  MoveL 1319 to (26.76, 68.08, -94.98) mm, rotated rx -9.61 ry -16.54 rz 125.97 deg; joints [-8.897, -67.323, 117.954, 201.647, 36.046, -119.29, -235]
  MoveL 1320 to (26.41, 68.69, -94.98) mm, rotated rx -9.61 ry -16.54 rz 125.97 deg; joints [-8.899, -67.37, 118.001, 201.644, 36.045, -119.288, -235]
  MoveL 1321 to (26.18, 69.29, -94.97) mm, rotated rx -9.61 ry -16.54 rz 125.97 deg; joints [-8.9, -67.415, 118.038, 201.646, 36.038, -119.292, -235]
  MoveL 1322 to (25.98, 69.92, -94.95) mm, rotated rx -9.61 ry -16.54 rz 125.97 deg; joints [-8.901, -67.462, 118.074, 201.65, 36.028, -119.298, -235]
  MoveL 1323 to (25.77, 70.66, -94.92) mm, rotated rx -9.61 ry -16.54 rz 125.97 deg; joints [-8.902, -67.516, 118.114, 201.657, 36.015, -119.306, -235]
  MoveL 1324 to (25.28, 72.7, -94.92) mm, rotated rx -9.61 ry -16.54 rz 125.97 deg; joints [-8.906, -67.664, 118.218, 201.672, 35.972, -119.329, -235]
  MoveL 1325 to (25.17, 73.13, -94.9) mm, rotated rx -9.61 ry -16.54 rz 125.97 deg; joints [-8.907, -67.696, 118.241, 201.676, 35.964, -119.335, -235]
  MoveL 1326 to (24.92, 74.15, -94.9) mm, rotated rx -9.61 ry -16.54 rz 125.97 deg; joints [-8.909, -67.77, 118.292, 201.684, 35.942, -119.347, -235]
  MoveL 1327 to (24.8, 74.64, -94.89) mm, rotated rx -9.61 ry -16.54 rz 125.97 deg; joints [-8.91, -67.806, 118.318, 201.688, 35.932, -119.352, -235]
  MoveL 1328 to (24.68, 75.11, -94.87) mm, rotated rx -9.61 ry -16.54 rz 125.97 deg; joints [-8.91, -67.841, 118.343, 201.692, 35.923, -119.358, -235]
  MoveL 1329 to (24.54, 75.57, -94.84) mm, rotated rx -9.61 ry -16.54 rz 125.97 deg; joints [-8.91, -67.875, 118.368, 201.697, 35.915, -119.364, -235]
  MoveL 1330 to (24.4, 75.98, -94.78) mm, rotated rx -9.61 ry -16.54 rz 125.97 deg; joints [-8.909, -67.906, 118.392, 201.703, 35.909, -119.37, -235]
  MoveL 1331 to (24.27, 76.44, -94.75) mm, rotated rx -9.61 ry -16.54 rz 125.97 deg; joints [-8.908, -67.939, 118.417, 201.708, 35.901, -119.376, -235]
  MoveL 1332 to (24.14, 76.91, -94.73) mm, rotated rx -9.61 ry -16.54 rz 125.97 deg; joints [-8.908, -67.974, 118.442, 201.712, 35.892, -119.381, -235]
  MoveL 1333 to (24.02, 77.41, -94.72) mm, rotated rx -9.61 ry -16.54 rz 125.97 deg; joints [-8.909, -68.01, 118.468, 201.717, 35.882, -119.387, -235]
  MoveL 1334 to (23.89, 77.88, -94.7) mm, rotated rx -9.61 ry -16.54 rz 125.97 deg; joints [-8.91, -68.045, 118.493, 201.721, 35.873, -119.393, -235]
  MoveL 1335 to (23.75, 78.34, -94.67) mm, rotated rx -9.61 ry -16.54 rz 125.97 deg; joints [-8.909, -68.079, 118.518, 201.726, 35.865, -119.399, -235]
  MoveL 1336 to (23.61, 78.75, -94.61) mm, rotated rx -9.61 ry -16.54 rz 125.97 deg; joints [-8.908, -68.11, 118.543, 201.731, 35.859, -119.404, -235]
  MoveL 1337 to (23.46, 79.18, -94.55) mm, rotated rx -9.61 ry -16.54 rz 125.97 deg; joints [-8.907, -68.143, 118.568, 201.737, 35.853, -119.41, -235]
  MoveL 1338 to (23.06, 80.57, -94.47) mm, rotated rx -9.61 ry -16.54 rz 125.97 deg; joints [-8.906, -68.245, 118.644, 201.751, 35.828, -119.427, -235]
  MoveL 1339 to (22.88, 81.73, -94.6) mm, rotated rx -9.61 ry -16.54 rz 125.97 deg; joints [-8.914, -68.328, 118.694, 201.755, 35.796, -119.44, -235]
  MoveL 1340 to (22.91, 82.67, -94.94) mm, rotated rx -9.61 ry -16.54 rz 125.97 deg; joints [-8.931, -68.392, 118.719, 201.749, 35.756, -119.448, -235]
  MoveL 1341 to (23.01, 83.06, -95.18) mm, rotated rx -9.61 ry -16.54 rz 125.97 deg; joints [-8.942, -68.416, 118.722, 201.742, 35.733, -119.45, -235]
  MoveL 1342 to (23.16, 83.39, -95.48) mm, rotated rx -9.61 ry -16.54 rz 125.97 deg; joints [-8.955, -68.436, 118.719, 201.733, 35.709, -119.451, -235]
  MoveL 1343 to (23.62, 83.9, -96.24) mm, rotated rx -9.61 ry -16.54 rz 125.97 deg; joints [-8.988, -68.461, 118.694, 201.706, 35.655, -119.449, -235]
  MoveL 1344 to (24.31, 84.18, -97.21) mm, rotated rx -9.61 ry -16.54 rz 125.97 deg; joints [-9.029, -68.466, 118.644, 201.669, 35.593, -119.443, -235]
  MoveL 1345 to (26.32, 84.09, -99.77) mm, rotated rx -9.61 ry -16.54 rz 125.97 deg; joints [-9.136, -68.419, 118.468, 201.565, 35.449, -119.415, -235]
  MoveL 1346 to (28.5, 83.24, -102.39) mm, rotated rx -9.61 ry -16.54 rz 125.97 deg; joints [-9.242, -68.314, 118.254, 201.451, 35.322, -119.375, -235]
  MoveL 1347 to (29.39, 82.56, -103.41) mm, rotated rx -9.61 ry -16.54 rz 125.97 deg; joints [-9.283, -68.249, 118.156, 201.402, 35.281, -119.353, -235]
  MoveL 1348 to (30.16, 81.72, -104.25) mm, rotated rx -9.61 ry -16.54 rz 125.97 deg; joints [-9.315, -68.176, 118.064, 201.358, 35.257, -119.33, -235]
  MoveL 1349 to (30.79, 80.72, -104.9) mm, rotated rx -9.61 ry -16.54 rz 125.97 deg; joints [-9.34, -68.094, 117.979, 201.32, 35.248, -119.307, -235]
  MoveL 1350 to (31.3, 79.55, -105.37) mm, rotated rx -9.61 ry -16.54 rz 125.97 deg; joints [-9.357, -68.004, 117.899, 201.288, 35.254, -119.283, -235]
  MoveL 1351 to (31.67, 78.22, -105.65) mm, rotated rx -9.61 ry -16.54 rz 125.97 deg; joints [-9.365, -67.905, 117.826, 201.261, 35.276, -119.258, -235]
  MoveL 1352 to (31.92, 76.73, -105.74) mm, rotated rx -9.61 ry -16.54 rz 125.97 deg; joints [-9.366, -67.798, 117.759, 201.239, 35.313, -119.232, -235]
  MoveL 1353 to (32.27, 73.59, -105.75) mm, rotated rx -9.61 ry -16.54 rz 125.97 deg; joints [-9.359, -67.576, 117.631, 201.203, 35.402, -119.181, -235]
  MoveL 1354 to (32.34, 73.04, -105.76) mm, rotated rx -9.61 ry -16.54 rz 125.97 deg; joints [-9.358, -67.537, 117.608, 201.196, 35.417, -119.172, -235]
  MoveL 1355 to (32.44, 72.42, -105.8) mm, rotated rx -9.61 ry -16.54 rz 125.97 deg; joints [-9.358, -67.493, 117.58, 201.187, 35.432, -119.161, -235]
  MoveL 1356 to (32.58, 71.68, -105.89) mm, rotated rx -9.61 ry -16.54 rz 125.97 deg; joints [-9.361, -67.439, 117.544, 201.174, 35.449, -119.148, -235]
  MoveL 1357 to (32.68, 71.07, -105.93) mm, rotated rx -9.61 ry -16.54 rz 125.97 deg; joints [-9.361, -67.395, 117.517, 201.166, 35.464, -119.137, -235]
  MoveL 1358 to (32.75, 70.53, -105.94) mm, rotated rx -9.61 ry -16.54 rz 125.97 deg; joints [-9.36, -67.357, 117.494, 201.159, 35.478, -119.128, -235]
  MoveL 1359 to (32.81, 70.02, -105.95) mm, rotated rx -9.61 ry -16.54 rz 125.97 deg; joints [-9.36, -67.321, 117.473, 201.153, 35.492, -119.12, -235]
  MoveL 1360 to (32.88, 69.57, -105.97) mm, rotated rx -9.61 ry -16.54 rz 125.97 deg; joints [-9.359, -67.289, 117.453, 201.147, 35.504, -119.113, -235]
  MoveL 1361 to (33.12, 67.53, -105.97) mm, rotated rx -9.61 ry -16.54 rz 125.97 deg; joints [-9.355, -67.145, 117.368, 201.124, 35.56, -119.08, -235]
  MoveL 1362 to (33.2, 67.02, -106.01) mm, rotated rx -9.61 ry -16.54 rz 125.97 deg; joints [-9.355, -67.109, 117.345, 201.117, 35.572, -119.072, -235]
  MoveL 1363 to (33.29, 66.56, -106.06) mm, rotated rx -9.61 ry -16.54 rz 125.97 deg; joints [-9.356, -67.075, 117.323, 201.109, 35.582, -119.064, -235]
  MoveL 1364 to (33.39, 66.11, -106.13) mm, rotated rx -9.61 ry -16.54 rz 125.97 deg; joints [-9.358, -67.042, 117.299, 201.101, 35.591, -119.056, -235]
  MoveL 1365 to (33.53, 65.64, -106.19) mm, rotated rx -9.61 ry -16.54 rz 125.97 deg; joints [-9.36, -67.008, 117.273, 201.095, 35.598, -119.049, -235]
  MoveL 1366 to (33.69, 65.11, -106.23) mm, rotated rx -9.61 ry -16.54 rz 125.97 deg; joints [-9.36, -66.969, 117.243, 201.091, 35.606, -119.044, -235]
  MoveL 1367 to (33.98, 64.51, -106.24) mm, rotated rx -9.61 ry -16.54 rz 125.97 deg; joints [-9.358, -66.923, 117.2, 201.092, 35.61, -119.043, -235]
  MoveL 1368 to (34.38, 63.84, -106.24) mm, rotated rx -9.61 ry -16.54 rz 125.97 deg; joints [-9.356, -66.871, 117.148, 201.096, 35.61, -119.046, -235]
  MoveL 1369 to (34.29, 65.78, -107.79) mm, rotated rx -9.61 ry -16.54 rz 125.97 deg; joints [-9.427, -66.999, 117.207, 201.017, 35.529, -119.016, -235]
  MoveL 1370 to (35.84, 64, -107.92) mm, rotated rx -9.61 ry -16.54 rz 125.97 deg; joints [-9.424, -66.852, 117.027, 201.037, 35.499, -119.039, -235]
  MoveL 1371 to (37.3, 62.31, -108.03) mm, rotated rx -9.61 ry -16.54 rz 125.97 deg; joints [-9.421, -66.713, 116.857, 201.058, 35.471, -119.061, -235]
  MoveL 1372 to (38.73, 60.68, -108.19) mm, rotated rx -9.61 ry -16.54 rz 125.97 deg; joints [-9.42, -66.579, 116.692, 201.075, 35.442, -119.082, -235]
  MoveL 1373 to (40.12, 59.07, -108.3) mm, rotated rx -9.61 ry -16.54 rz 125.97 deg; joints [-9.418, -66.446, 116.529, 201.095, 35.414, -119.103, -235]
  MoveL 1374 to (41.52, 57.45, -108.41) mm, rotated rx -9.61 ry -16.54 rz 125.97 deg; joints [-9.415, -66.313, 116.365, 201.114, 35.386, -119.125, -235]
  MoveL 1375 to (42.92, 55.84, -108.63) mm, rotated rx -9.61 ry -16.54 rz 125.97 deg; joints [-9.417, -66.181, 116.201, 201.127, 35.356, -119.143, -235]
  MoveL 1376 to (44.32, 54.23, -108.86) mm, rotated rx -9.61 ry -16.54 rz 125.97 deg; joints [-9.419, -66.048, 116.036, 201.14, 35.326, -119.16, -235]
  MoveL 1377 to (45.71, 52.61, -108.97) mm, rotated rx -9.61 ry -16.54 rz 125.97 deg; joints [-9.416, -65.915, 115.872, 201.16, 35.298, -119.182, -235]
  MoveL 1378 to (47.09, 50.98, -108.97) mm, rotated rx -9.61 ry -16.54 rz 125.97 deg; joints [-9.409, -65.782, 115.71, 201.187, 35.272, -119.209, -235]
  MoveL 1379 to (48.48, 49.36, -109.08) mm, rotated rx -9.61 ry -16.54 rz 125.97 deg; joints [-9.406, -65.65, 115.546, 201.207, 35.243, -119.231, -235]
  MoveL 1380 to (49.88, 47.71, -109.29) mm, rotated rx -9.61 ry -16.54 rz 125.97 deg; joints [-9.408, -65.515, 115.379, 201.222, 35.213, -119.25, -235]
  MoveL 1381 to (51.19, 46.18, -109.47) mm, rotated rx -9.61 ry -16.54 rz 125.97 deg; joints [-9.408, -65.389, 115.223, 201.236, 35.185, -119.268, -235]
  MoveL 1382 to (52.39, 44.76, -109.68) mm, rotated rx -9.61 ry -16.54 rz 125.97 deg; joints [-9.411, -65.273, 115.079, 201.246, 35.158, -119.282, -235]
  MoveL 1383 to (53.66, 43.26, -109.77) mm, rotated rx -9.61 ry -16.54 rz 125.97 deg; joints [-9.408, -65.151, 114.928, 201.266, 35.131, -119.304, -235]
  MoveL 1384 to (55.01, 41.67, -109.79) mm, rotated rx -9.61 ry -16.54 rz 125.97 deg; joints [-9.402, -65.021, 114.767, 201.292, 35.104, -119.331, -235]
  MoveL 1385 to (56.75, 39.59, -109.88) mm, rotated rx -9.61 ry -16.54 rz 125.97 deg; joints [-9.397, -64.853, 114.558, 201.322, 35.067, -119.361, -235]
  MoveL 1386 to (58.05, 38.03, -110.1) mm, rotated rx -9.61 ry -16.54 rz 125.97 deg; joints [-9.399, -64.725, 114.4, 201.334, 35.039, -119.378, -235]
  MoveL 1387 to (59.45, 36.33, -110.3) mm, rotated rx -9.61 ry -16.54 rz 125.97 deg; joints [-9.4, -64.587, 114.23, 201.349, 35.008, -119.398, -235]
  MoveL 1388 to (60.73, 34.76, -110.58) mm, rotated rx -9.61 ry -16.54 rz 125.97 deg; joints [-9.405, -64.46, 114.073, 201.356, 34.979, -119.411, -235]
  MoveL 1389 to (62, 33.24, -110.71) mm, rotated rx -9.61 ry -16.54 rz 125.97 deg; joints [-9.404, -64.336, 113.919, 201.374, 34.951, -119.432, -235]
  MoveL 1390 to (63.36, 31.64, -110.73) mm, rotated rx -9.61 ry -16.54 rz 125.97 deg; joints [-9.397, -64.207, 113.756, 201.402, 34.922, -119.46, -235]
  MoveL 1391 to (64.46, 30.25, -110.96) mm, rotated rx -9.61 ry -16.54 rz 125.97 deg; joints [-9.401, -64.095, 113.619, 201.409, 34.897, -119.472, -235]
  Set speed (1000.0 mm/s)
  MoveL 1392 to (88.08, 19.24, -110.96) mm, rotated rx -9.61 ry -16.54 rz 125.97 deg; joints [-9.309, -62.966, 111.351, 202.177, 33.862, -120.32, -235]
  Set speed (1000.0 mm/s)
  MoveL 1393 to (85.31, 13.32, -122.15) mm, rotated rx -9.61 ry -16.54 rz 125.97 deg; joints [-9.767, -62.572, 111.273, 201.243, 34.045, -119.606, -235]
  Set speed (100.0 mm/s)
  MoveL 1394 to (67.03, 21.84, -122.15) mm, rotated rx -9.61 ry -16.54 rz 125.97 deg; joints [-9.843, -63.44, 113.032, 200.653, 34.858, -118.961, -235]
  MoveL 1395 to (65.87, 23.63, -122.15) mm, rotated rx -9.61 ry -16.54 rz 125.97 deg; joints [-9.851, -63.579, 113.188, 200.632, 34.872, -118.942, -235]
  MoveL 1396 to (64.67, 25.51, -122.05) mm, rotated rx -9.61 ry -16.54 rz 125.97 deg; joints [-9.855, -63.725, 113.35, 200.618, 34.886, -118.929, -235]
  MoveL 1397 to (63.44, 27.51, -121.75) mm, rotated rx -9.61 ry -16.54 rz 125.97 deg; joints [-9.85, -63.88, 113.52, 200.617, 34.901, -118.924, -235]
  MoveL 1398 to (62.26, 29.43, -121.41) mm, rotated rx -9.61 ry -16.54 rz 125.97 deg; joints [-9.844, -64.03, 113.683, 200.621, 34.915, -118.923, -235]
  MoveL 1399 to (61.15, 31.18, -121.22) mm, rotated rx -9.61 ry -16.54 rz 125.97 deg; joints [-9.843, -64.166, 113.833, 200.616, 34.928, -118.915, -235]
  MoveL 1400 to (60.1, 32.82, -121.08) mm, rotated rx -9.61 ry -16.54 rz 125.97 deg; joints [-9.844, -64.294, 113.974, 200.607, 34.941, -118.906, -235]
  MoveL 1401 to (58.98, 34.54, -121.03) mm, rotated rx -9.61 ry -16.54 rz 125.97 deg; joints [-9.849, -64.428, 114.123, 200.592, 34.953, -118.892, -235]
  MoveL 1402 to (57.82, 36.33, -121.01) mm, rotated rx -9.61 ry -16.54 rz 125.97 deg; joints [-9.856, -64.567, 114.277, 200.573, 34.965, -118.876, -235]
  MoveL 1403 to (56.66, 38.11, -120.89) mm, rotated rx -9.61 ry -16.54 rz 125.97 deg; joints [-9.858, -64.706, 114.43, 200.562, 34.978, -118.864, -235]
  MoveL 1404 to (55.42, 40.03, -120.63) mm, rotated rx -9.61 ry -16.54 rz 125.97 deg; joints [-9.856, -64.857, 114.596, 200.559, 34.992, -118.858, -235]
  MoveL 1405 to (54.1, 42.04, -120.45) mm, rotated rx -9.61 ry -16.54 rz 125.97 deg; joints [-9.856, -65.015, 114.769, 200.55, 35.007, -118.847, -235]
  MoveL 1406 to (52.82, 43.99, -120.25) mm, rotated rx -9.61 ry -16.54 rz 125.97 deg; joints [-9.856, -65.168, 114.938, 200.543, 35.022, -118.838, -235]
  MoveL 1407 to (51.65, 45.77, -120.13) mm, rotated rx -9.61 ry -16.54 rz 125.97 deg; joints [-9.859, -65.308, 115.092, 200.531, 35.034, -118.827, -235]
  MoveL 1408 to (49.32, 49.29, -119.86) mm, rotated rx -9.61 ry -16.54 rz 125.97 deg; joints [-9.862, -65.585, 115.396, 200.512, 35.058, -118.807, -235]
  MoveL 1409 to (48.13, 51.11, -119.79) mm, rotated rx -9.61 ry -16.54 rz 125.97 deg; joints [-9.867, -65.728, 115.551, 200.498, 35.068, -118.794, -235]
  MoveL 1410 to (46.94, 52.88, -119.57) mm, rotated rx -9.61 ry -16.54 rz 125.97 deg; joints [-9.866, -65.868, 115.705, 200.494, 35.082, -118.787, -235]
  MoveL 1411 to (45.76, 54.63, -119.41) mm, rotated rx -9.61 ry -16.54 rz 125.97 deg; joints [-9.866, -66.007, 115.857, 200.486, 35.094, -118.778, -235]
  MoveL 1412 to (44.58, 56.38, -119.23) mm, rotated rx -9.61 ry -16.54 rz 125.97 deg; joints [-9.866, -66.146, 116.009, 200.479, 35.107, -118.77, -235]
  MoveL 1413 to (43.37, 58.2, -119.14) mm, rotated rx -9.61 ry -16.54 rz 125.97 deg; joints [-9.87, -66.289, 116.164, 200.467, 35.117, -118.759, -235]
  MoveL 1414 to (42.1, 60.08, -119.01) mm, rotated rx -9.61 ry -16.54 rz 125.97 deg; joints [-9.873, -66.438, 116.327, 200.456, 35.13, -118.748, -235]
  MoveL 1415 to (41.06, 61.67, -118.95) mm, rotated rx -9.61 ry -16.54 rz 125.97 deg; joints [-9.877, -66.564, 116.461, 200.445, 35.136, -118.738, -235]
  MoveL 1416 to (40.5, 61.31, -118.06) mm, rotated rx -9.61 ry -16.54 rz 125.97 deg; joints [-9.84, -66.551, 116.499, 200.479, 35.192, -118.746, -235]
  MoveL 1417 to (40.48, 60.95, -117.65) mm, rotated rx -9.61 ry -16.54 rz 125.97 deg; joints [-9.822, -66.529, 116.492, 200.502, 35.21, -118.756, -235]
  MoveL 1418 to (40.44, 60.9, -117.37) mm, rotated rx -9.61 ry -16.54 rz 125.97 deg; joints [-9.81, -66.527, 116.496, 200.518, 35.218, -118.765, -235]
  MoveL 1419 to (40.39, 61.22, -117.26) mm, rotated rx -9.61 ry -16.54 rz 125.97 deg; joints [-9.806, -66.551, 116.511, 200.529, 35.212, -118.774, -235]
  MoveL 1420 to (40.36, 61.67, -117.19) mm, rotated rx -9.61 ry -16.54 rz 125.97 deg; joints [-9.804, -66.582, 116.529, 200.538, 35.199, -118.785, -235]
  MoveL 1421 to (40.34, 62.23, -117.16) mm, rotated rx -9.61 ry -16.54 rz 125.97 deg; joints [-9.804, -66.621, 116.549, 200.548, 35.182, -118.796, -235]
  MoveL 1422 to (40.33, 62.93, -117.12) mm, rotated rx -9.61 ry -16.54 rz 125.97 deg; joints [-9.804, -66.669, 116.574, 200.56, 35.16, -118.811, -235]
  MoveL 1423 to (40.32, 63.56, -117.1) mm, rotated rx -9.61 ry -16.54 rz 125.97 deg; joints [-9.804, -66.712, 116.595, 200.571, 35.139, -118.824, -235]
  MoveL 1424 to (40.33, 64.08, -117.1) mm, rotated rx -9.61 ry -16.54 rz 125.97 deg; joints [-9.805, -66.748, 116.612, 200.579, 35.121, -118.835, -235]
  MoveL 1425 to (40.32, 64.57, -117.08) mm, rotated rx -9.61 ry -16.54 rz 125.97 deg; joints [-9.805, -66.782, 116.628, 200.587, 35.105, -118.845, -235]
  MoveL 1426 to (40.28, 65.61, -117) mm, rotated rx -9.61 ry -16.54 rz 125.97 deg; joints [-9.804, -66.854, 116.666, 200.606, 35.073, -118.867, -235]
  MoveL 1427 to (40.25, 66.17, -116.95) mm, rotated rx -9.61 ry -16.54 rz 125.97 deg; joints [-9.803, -66.893, 116.687, 200.616, 35.056, -118.879, -235]
  MoveL 1428 to (40.21, 66.68, -116.89) mm, rotated rx -9.61 ry -16.54 rz 125.97 deg; joints [-9.802, -66.928, 116.707, 200.627, 35.042, -118.89, -235]
  MoveL 1429 to (40.17, 67.14, -116.81) mm, rotated rx -9.61 ry -16.54 rz 125.97 deg; joints [-9.8, -66.961, 116.726, 200.637, 35.03, -118.901, -235]
  MoveL 1430 to (40.14, 67.6, -116.75) mm, rotated rx -9.61 ry -16.54 rz 125.97 deg; joints [-9.798, -66.994, 116.744, 200.647, 35.016, -118.911, -235]
  MoveL 1431 to (40.12, 68.09, -116.72) mm, rotated rx -9.61 ry -16.54 rz 125.97 deg; joints [-9.798, -67.027, 116.761, 200.655, 35.001, -118.922, -235]
  MoveL 1432 to (40.11, 68.61, -116.7) mm, rotated rx -9.61 ry -16.54 rz 125.97 deg; joints [-9.798, -67.063, 116.779, 200.664, 34.984, -118.933, -235]
  MoveL 1433 to (40.15, 72.28, -116.7) mm, rotated rx -9.61 ry -16.54 rz 125.97 deg; joints [-9.805, -67.313, 116.893, 200.721, 34.856, -119.009, -235]
  MoveL 1434 to (40.28, 73.9, -116.72) mm, rotated rx -9.61 ry -16.54 rz 125.97 deg; joints [-9.809, -67.422, 116.935, 200.749, 34.792, -119.046, -235]
  MoveL 1435 to (40.42, 74.46, -116.75) mm, rotated rx -9.61 ry -16.54 rz 125.97 deg; joints [-9.811, -67.458, 116.942, 200.761, 34.765, -119.062, -235]
  MoveL 1436 to (40.6, 74.86, -116.78) mm, rotated rx -9.61 ry -16.54 rz 125.97 deg; joints [-9.813, -67.482, 116.941, 200.771, 34.74, -119.076, -235]
  MoveL 1437 to (40.81, 75.13, -116.83) mm, rotated rx -9.61 ry -16.54 rz 125.97 deg; joints [-9.814, -67.497, 116.932, 200.78, 34.718, -119.089, -235]
  MoveL 1438 to (40.93, 75.21, -116.85) mm, rotated rx -9.61 ry -16.54 rz 125.97 deg; joints [-9.815, -67.5, 116.925, 200.784, 34.708, -119.095, -235]
  MoveL 1439 to (41.06, 75.26, -116.87) mm, rotated rx -9.61 ry -16.54 rz 125.97 deg; joints [-9.816, -67.502, 116.916, 200.788, 34.698, -119.1, -235]
  MoveL 1440 to (41.2, 75.28, -116.9) mm, rotated rx -9.61 ry -16.54 rz 125.97 deg; joints [-9.816, -67.501, 116.906, 200.792, 34.69, -119.105, -235]
  MoveL 1441 to (41.34, 75.28, -116.93) mm, rotated rx -9.61 ry -16.54 rz 125.97 deg; joints [-9.817, -67.498, 116.895, 200.795, 34.681, -119.11, -235]
  MoveL 1442 to (41.65, 75.19, -116.99) mm, rotated rx -9.61 ry -16.54 rz 125.97 deg; joints [-9.819, -67.487, 116.868, 200.801, 34.666, -119.118, -235]
  MoveL 1443 to (42.31, 74.76, -117.12) mm, rotated rx -9.61 ry -16.54 rz 125.97 deg; joints [-9.821, -67.445, 116.801, 200.81, 34.642, -119.132, -235]
  MoveL 1444 to (43.02, 74.05, -117.26) mm, rotated rx -9.61 ry -16.54 rz 125.97 deg; joints [-9.823, -67.385, 116.721, 200.816, 34.624, -119.141, -235]
  MoveL 1445 to (44.45, 72.19, -117.53) mm, rotated rx -9.61 ry -16.54 rz 125.97 deg; joints [-9.826, -67.233, 116.548, 200.823, 34.603, -119.152, -235]
  MoveL 1446 to (45.79, 70.18, -117.77) mm, rotated rx -9.61 ry -16.54 rz 125.97 deg; joints [-9.828, -67.073, 116.377, 200.826, 34.592, -119.157, -235]
  MoveL 1447 to (75.46, 25.08, -122.85) mm, rotated rx -9.61 ry -16.54 rz 125.97 deg; joints [-9.851, -63.517, 112.474, 200.968, 34.262, -119.351, -235]
  MoveL 1448 to (77.56, 21.88, -123.22) mm, rotated rx -9.61 ry -16.54 rz 125.97 deg; joints [-9.853, -63.267, 112.19, 200.983, 34.231, -119.37, -235]
  MoveL 1449 to (79.47, 18.65, -123.63) mm, rotated rx -9.61 ry -16.54 rz 125.97 deg; joints [-9.857, -63.018, 111.92, 200.986, 34.21, -119.379, -235]
  MoveL 1450 to (79.98, 17.25, -123.84) mm, rotated rx -9.61 ry -16.54 rz 125.97 deg; joints [-9.861, -62.915, 111.827, 200.974, 34.218, -119.367, -235]
  MoveL 1451 to (80.02, 16.7, -123.94) mm, rotated rx -9.61 ry -16.54 rz 125.97 deg; joints [-9.864, -62.877, 111.804, 200.962, 34.231, -119.356, -235]
  MoveL 1452 to (79.97, 16.48, -123.98) mm, rotated rx -9.61 ry -16.54 rz 125.97 deg; joints [-9.866, -62.863, 111.799, 200.954, 34.24, -119.348, -235]
  MoveL 1453 to (79.87, 16.3, -124.02) mm, rotated rx -9.61 ry -16.54 rz 125.97 deg; joints [-9.867, -62.852, 111.8, 200.945, 34.25, -119.338, -235]
  MoveL 1454 to (79.71, 16.16, -124.06) mm, rotated rx -9.61 ry -16.54 rz 125.97 deg; joints [-9.869, -62.845, 111.807, 200.935, 34.263, -119.328, -235]
  MoveL 1455 to (79.5, 16.06, -124.09) mm, rotated rx -9.61 ry -16.54 rz 125.97 deg; joints [-9.871, -62.842, 111.82, 200.924, 34.277, -119.315, -235]
  MoveL 1456 to (79.23, 16.02, -124.12) mm, rotated rx -9.61 ry -16.54 rz 125.97 deg; joints [-9.873, -62.844, 111.84, 200.91, 34.294, -119.301, -235]
  MoveL 1457 to (78.89, 16.03, -124.15) mm, rotated rx -9.61 ry -16.54 rz 125.97 deg; joints [-9.875, -62.85, 111.868, 200.896, 34.314, -119.285, -235]
  MoveL 1458 to (76.79, 16.66, -124.2) mm, rotated rx -9.61 ry -16.54 rz 125.97 deg; joints [-9.886, -62.926, 112.057, 200.82, 34.417, -119.203, -235]
  MoveL 1459 to (74.86, 17.48, -124.2) mm, rotated rx -9.61 ry -16.54 rz 125.97 deg; joints [-9.894, -63.013, 112.24, 200.757, 34.505, -119.134, -235]
  MoveL 1460 to (71.56, 19.38, -124.24) mm, rotated rx -9.61 ry -16.54 rz 125.97 deg; joints [-9.91, -63.193, 112.569, 200.653, 34.64, -119.023, -235]
  MoveL 1461 to (68.95, 21.77, -124.35) mm, rotated rx -9.61 ry -16.54 rz 125.97 deg; joints [-9.929, -63.395, 112.86, 200.578, 34.72, -118.949, -235]
  MoveL 1462 to (65.63, 26.83, -124.65) mm, rotated rx -9.61 ry -16.54 rz 125.97 deg; joints [-9.963, -63.786, 113.3, 200.498, 34.757, -118.883, -235]
  MoveL 1463 to (64.77, 29.03, -124.78) mm, rotated rx -9.61 ry -16.54 rz 125.97 deg; joints [-9.975, -63.947, 113.444, 200.485, 34.738, -118.879, -235]
  MoveL 1464 to (53.51, 61.93, -126.65) mm, rotated rx -9.61 ry -16.54 rz 125.97 deg; joints [-10.163, -66.343, 115.431, 200.383, 34.313, -118.928, -235]
  MoveL 1465 to (52.54, 64.74, -126.81) mm, rotated rx -9.61 ry -16.54 rz 125.97 deg; joints [-10.18, -66.549, 115.598, 200.376, 34.273, -118.934, -235]
  MoveL 1466 to (50.89, 68.09, -127.05) mm, rotated rx -9.61 ry -16.54 rz 125.97 deg; joints [-10.203, -66.802, 115.834, 200.345, 34.251, -118.919, -235]
  MoveL 1467 to (49.96, 69.24, -127.19) mm, rotated rx -9.61 ry -16.54 rz 125.97 deg; joints [-10.215, -66.895, 115.943, 200.317, 34.263, -118.896, -235]
  MoveL 1468 to (49.5, 69.55, -127.26) mm, rotated rx -9.61 ry -16.54 rz 125.97 deg; joints [-10.221, -66.923, 115.988, 200.3, 34.278, -118.88, -235]
  MoveL 1469 to (49.29, 69.61, -127.3) mm, rotated rx -9.61 ry -16.54 rz 125.97 deg; joints [-10.223, -66.931, 116.007, 200.29, 34.288, -118.87, -235]
  MoveL 1470 to (49.08, 69.62, -127.33) mm, rotated rx -9.61 ry -16.54 rz 125.97 deg; joints [-10.226, -66.935, 116.023, 200.28, 34.299, -118.86, -235]
  MoveL 1471 to (48.88, 69.55, -127.37) mm, rotated rx -9.61 ry -16.54 rz 125.97 deg; joints [-10.228, -66.934, 116.036, 200.269, 34.312, -118.849, -235]
  MoveL 1472 to (48.69, 69.41, -127.4) mm, rotated rx -9.61 ry -16.54 rz 125.97 deg; joints [-10.229, -66.927, 116.046, 200.258, 34.327, -118.837, -235]
  MoveL 1473 to (48.51, 69.19, -127.44) mm, rotated rx -9.61 ry -16.54 rz 125.97 deg; joints [-10.231, -66.915, 116.053, 200.246, 34.344, -118.824, -235]
  MoveL 1474 to (48.35, 68.89, -127.47) mm, rotated rx -9.61 ry -16.54 rz 125.97 deg; joints [-10.232, -66.897, 116.056, 200.233, 34.364, -118.809, -235]
  MoveL 1475 to (47.87, 66.75, -127.59) mm, rotated rx -9.61 ry -16.54 rz 125.97 deg; joints [-10.235, -66.759, 116.023, 200.176, 34.462, -118.742, -235]
  MoveL 1476 to (47.81, 66.24, -127.61) mm, rotated rx -9.61 ry -16.54 rz 125.97 deg; joints [-10.235, -66.725, 116.011, 200.165, 34.483, -118.729, -235]
  MoveL 1477 to (47.79, 65.78, -127.66) mm, rotated rx -9.61 ry -16.54 rz 125.97 deg; joints [-10.236, -66.694, 115.998, 200.154, 34.499, -118.717, -235]
  MoveL 1478 to (47.78, 65.34, -127.73) mm, rotated rx -9.61 ry -16.54 rz 125.97 deg; joints [-10.238, -66.663, 115.983, 200.143, 34.513, -118.705, -235]
  MoveL 1479 to (47.76, 64.89, -127.79) mm, rotated rx -9.61 ry -16.54 rz 125.97 deg; joints [-10.239, -66.633, 115.97, 200.132, 34.529, -118.693, -235]
  MoveL 1480 to (47.73, 64.43, -127.82) mm, rotated rx -9.61 ry -16.54 rz 125.97 deg; joints [-10.24, -66.602, 115.957, 200.122, 34.546, -118.682, -235]
  MoveL 1481 to (47.09, 59.79, -127.83) mm, rotated rx -9.61 ry -16.54 rz 125.97 deg; joints [-10.233, -66.297, 115.855, 200.033, 34.739, -118.567, -235]
  MoveL 1482 to (47.04, 59.35, -127.86) mm, rotated rx -9.61 ry -16.54 rz 125.97 deg; joints [-10.233, -66.268, 115.844, 200.024, 34.756, -118.556, -235]
  MoveL 1483 to (46.98, 58.88, -127.87) mm, rotated rx -9.61 ry -16.54 rz 125.97 deg; joints [-10.232, -66.237, 115.833, 200.014, 34.775, -118.544, -235]
  MoveL 1484 to (46.84, 57.85, -127.87) mm, rotated rx -9.61 ry -16.54 rz 125.97 deg; joints [-10.231, -66.169, 115.81, 199.995, 34.817, -118.519, -235]
  MoveL 1485 to (46.77, 57.28, -127.88) mm, rotated rx -9.61 ry -16.54 rz 125.97 deg; joints [-10.23, -66.131, 115.797, 199.984, 34.84, -118.505, -235]
  MoveL 1486 to (46.72, 56.68, -127.89) mm, rotated rx -9.61 ry -16.54 rz 125.97 deg; joints [-10.23, -66.091, 115.781, 199.973, 34.863, -118.491, -235]
  MoveL 1487 to (46.7, 56.02, -127.92) mm, rotated rx -9.61 ry -16.54 rz 125.97 deg; joints [-10.229, -66.047, 115.76, 199.962, 34.885, -118.477, -235]
  MoveL 1488 to (46.76, 55.36, -127.95) mm, rotated rx -9.61 ry -16.54 rz 125.97 deg; joints [-10.229, -66.001, 115.733, 199.953, 34.904, -118.466, -235]
  MoveL 1489 to (46.87, 54.72, -127.96) mm, rotated rx -9.61 ry -16.54 rz 125.97 deg; joints [-10.228, -65.955, 115.703, 199.948, 34.918, -118.458, -235]
  MoveL 1490 to (46.94, 56.03, -128.94) mm, rotated rx -9.61 ry -16.54 rz 125.97 deg; joints [-10.272, -66.038, 115.733, 199.901, 34.858, -118.443, -235]
  MoveL 1491 to (47.8, 55, -129.37) mm, rotated rx -9.61 ry -16.54 rz 125.97 deg; joints [-10.285, -65.952, 115.628, 199.89, 34.837, -118.441, -235]
  MoveL 1492 to (48.64, 53.77, -129.69) mm, rotated rx -9.61 ry -16.54 rz 125.97 deg; joints [-10.293, -65.854, 115.518, 199.882, 34.825, -118.439, -235]
  MoveL 1493 to (49.5, 52.31, -129.92) mm, rotated rx -9.61 ry -16.54 rz 125.97 deg; joints [-10.296, -65.74, 115.4, 199.879, 34.82, -118.438, -235]
  MoveL 1494 to (50.48, 50.41, -130.14) mm, rotated rx -9.61 ry -16.54 rz 125.97 deg; joints [-10.297, -65.594, 115.258, 199.875, 34.823, -118.435, -235]
  MoveL 1495 to (51.43, 48.5, -130.25) mm, rotated rx -9.61 ry -16.54 rz 125.97 deg; joints [-10.295, -65.449, 115.118, 199.877, 34.829, -118.435, -235]
  MoveL 1496 to (52.38, 46.59, -130.36) mm, rotated rx -9.61 ry -16.54 rz 125.97 deg; joints [-10.291, -65.304, 114.977, 199.88, 34.834, -118.435, -235]
  MoveL 1497 to (53.35, 44.68, -130.59) mm, rotated rx -9.61 ry -16.54 rz 125.97 deg; joints [-10.293, -65.158, 114.835, 199.875, 34.837, -118.431, -235]
  MoveL 1498 to (54.29, 42.77, -130.71) mm, rotated rx -9.61 ry -16.54 rz 125.97 deg; joints [-10.291, -65.013, 114.695, 199.877, 34.842, -118.431, -235]
  MoveL 1499 to (55.24, 40.86, -130.94) mm, rotated rx -9.61 ry -16.54 rz 125.97 deg; joints [-10.293, -64.868, 114.553, 199.872, 34.844, -118.427, -235]
  MoveL 1500 to (56.18, 38.95, -131.06) mm, rotated rx -9.61 ry -16.54 rz 125.97 deg; joints [-10.29, -64.723, 114.412, 199.874, 34.849, -118.427, -235]
  MoveL 1501 to (57.12, 37.03, -131.18) mm, rotated rx -9.61 ry -16.54 rz 125.97 deg; joints [-10.287, -64.578, 114.271, 199.877, 34.853, -118.428, -235]
  MoveL 1502 to (58.06, 35.11, -131.41) mm, rotated rx -9.61 ry -16.54 rz 125.97 deg; joints [-10.29, -64.432, 114.129, 199.871, 34.856, -118.423, -235]
  MoveL 1503 to (58.94, 33.27, -131.52) mm, rotated rx -9.61 ry -16.54 rz 125.97 deg; joints [-10.287, -64.294, 113.995, 199.874, 34.861, -118.424, -235]
  MoveL 1504 to (59.79, 31.48, -131.72) mm, rotated rx -9.61 ry -16.54 rz 125.97 deg; joints [-10.288, -64.158, 113.863, 199.87, 34.864, -118.42, -235]
  MoveL 1505 to (60.84, 29.35, -131.88) mm, rotated rx -9.61 ry -16.54 rz 125.97 deg; joints [-10.287, -63.998, 113.705, 199.871, 34.867, -118.42, -235]
  MoveL 1506 to (62, 26.89, -131.97) mm, rotated rx -9.61 ry -16.54 rz 125.97 deg; joints [-10.281, -63.813, 113.526, 199.878, 34.873, -118.423, -235]
  MoveL 1507 to (62.9, 25.02, -132.04) mm, rotated rx -9.61 ry -16.54 rz 125.97 deg; joints [-10.276, -63.673, 113.388, 199.884, 34.877, -118.426, -235]
  MoveL 1508 to (63.74, 23.28, -132.17) mm, rotated rx -9.61 ry -16.54 rz 125.97 deg; joints [-10.275, -63.542, 113.259, 199.886, 34.879, -118.427, -235]
  MoveL 1509 to (64.6, 21.5, -132.27) mm, rotated rx -9.61 ry -16.54 rz 125.97 deg; joints [-10.272, -63.408, 113.127, 199.889, 34.881, -118.429, -235]
  MoveL 1510 to (65.44, 19.73, -132.38) mm, rotated rx -9.61 ry -16.54 rz 125.97 deg; joints [-10.27, -63.276, 112.997, 199.892, 34.883, -118.43, -235]
  MoveL 1511 to (66.33, 17.88, -132.45) mm, rotated rx -9.61 ry -16.54 rz 125.97 deg; joints [-10.266, -63.137, 112.859, 199.898, 34.886, -118.433, -235]
  MoveL 1512 to (67.28, 15.87, -132.55) mm, rotated rx -9.61 ry -16.54 rz 125.97 deg; joints [-10.262, -62.987, 112.711, 199.903, 34.888, -118.436, -235]
  MoveL 1513 to (68.29, 13.68, -132.81) mm, rotated rx -9.61 ry -16.54 rz 125.97 deg; joints [-10.265, -62.823, 112.55, 199.898, 34.89, -118.432, -235]
  MoveL 1514 to (69.67, 11.92, -133.8) mm, rotated rx -9.61 ry -16.54 rz 125.97 deg; joints [-10.296, -62.678, 112.368, 199.864, 34.848, -118.42, -235]
  MoveL 1515 to (68.7, 12.51, -134.28) mm, rotated rx -9.61 ry -16.54 rz 125.97 deg; joints [-10.321, -62.731, 112.462, 199.803, 34.882, -118.369, -235]
  MoveL 1516 to (68.18, 12.81, -134.59) mm, rotated rx -9.61 ry -16.54 rz 125.97 deg; joints [-10.337, -62.758, 112.511, 199.767, 34.9, -118.339, -235]
  MoveL 1517 to (68.09, 12.86, -134.74) mm, rotated rx -9.61 ry -16.54 rz 125.97 deg; joints [-10.343, -62.761, 112.518, 199.754, 34.901, -118.33, -235]
  MoveL 1518 to (68.39, 12.68, -134.78) mm, rotated rx -9.61 ry -16.54 rz 125.97 deg; joints [-10.343, -62.744, 112.488, 199.761, 34.889, -118.338, -235]
  MoveL 1519 to (68.79, 12.44, -134.8) mm, rotated rx -9.61 ry -16.54 rz 125.97 deg; joints [-10.342, -62.722, 112.448, 199.772, 34.872, -118.35, -235]
  MoveL 1520 to (69.19, 12.18, -134.83) mm, rotated rx -9.61 ry -16.54 rz 125.97 deg; joints [-10.341, -62.698, 112.406, 199.781, 34.856, -118.361, -235]
  MoveL 1521 to (69.56, 11.92, -134.89) mm, rotated rx -9.61 ry -16.54 rz 125.97 deg; joints [-10.342, -62.675, 112.367, 199.788, 34.841, -118.37, -235]
  MoveL 1522 to (69.95, 11.67, -134.93) mm, rotated rx -9.61 ry -16.54 rz 125.97 deg; joints [-10.342, -62.651, 112.327, 199.796, 34.825, -118.38, -235]
  MoveL 1523 to (70.37, 11.41, -134.95) mm, rotated rx -9.61 ry -16.54 rz 125.97 deg; joints [-10.34, -62.627, 112.285, 199.808, 34.808, -118.393, -235]
  MoveL 1524 to (72.63, 10.09, -134.95) mm, rotated rx -9.61 ry -16.54 rz 125.97 deg; joints [-10.329, -62.503, 112.057, 199.876, 34.713, -118.466, -235]
  MoveL 1525 to (73.02, 9.85, -134.97) mm, rotated rx -9.61 ry -16.54 rz 125.97 deg; joints [-10.328, -62.481, 112.018, 199.886, 34.697, -118.477, -235]
  MoveL 1526 to (73.34, 9.63, -135.01) mm, rotated rx -9.61 ry -16.54 rz 125.97 deg; joints [-10.328, -62.461, 111.984, 199.894, 34.684, -118.486, -235]
  MoveL 1527 to (73.73, 9.39, -135.03) mm, rotated rx -9.61 ry -16.54 rz 125.97 deg; joints [-10.327, -62.439, 111.944, 199.904, 34.668, -118.497, -235]
  MoveL 1528 to (74.24, 9.07, -135.05) mm, rotated rx -9.61 ry -16.54 rz 125.97 deg; joints [-10.325, -62.409, 111.892, 199.918, 34.647, -118.513, -235]
  MoveL 1529 to (74.84, 8.67, -135.1) mm, rotated rx -9.61 ry -16.54 rz 125.97 deg; joints [-10.325, -62.373, 111.829, 199.932, 34.622, -118.529, -235]
  MoveL 1530 to (75.36, 8.35, -135.13) mm, rotated rx -9.61 ry -16.54 rz 125.97 deg; joints [-10.323, -62.343, 111.775, 199.946, 34.601, -118.545, -235]
  MoveL 1531 to (75.82, 8.08, -135.13) mm, rotated rx -9.61 ry -16.54 rz 125.97 deg; joints [-10.321, -62.317, 111.729, 199.96, 34.581, -118.56, -235]
  MoveL 1532 to (77.18, 7.28, -135.13) mm, rotated rx -9.61 ry -16.54 rz 125.97 deg; joints [-10.315, -62.243, 111.592, 200.001, 34.524, -118.604, -235]
  MoveL 1533 to (79.54, 5.57, -135.48) mm, rotated rx -9.61 ry -16.54 rz 125.97 deg; joints [-10.316, -62.089, 111.339, 200.048, 34.431, -118.662, -235]
  MoveL 1534 to (80.42, 4.62, -135.9) mm, rotated rx -9.61 ry -16.54 rz 125.97 deg; joints [-10.329, -62.009, 111.23, 200.042, 34.4, -118.667, -235]
  MoveL 1535 to (81.12, 3.62, -136.5) mm, rotated rx -9.61 ry -16.54 rz 125.97 deg; joints [-10.349, -61.928, 111.132, 200.018, 34.38, -118.656, -235]
  MoveL 1536 to (81.93, 1.45, -138.21) mm, rotated rx -9.61 ry -16.54 rz 125.97 deg; joints [-10.411, -61.762, 110.972, 199.912, 34.372, -118.584, -235]
  MoveL 1537 to (81.96, -0.96, -140.61) mm, rotated rx -9.61 ry -16.54 rz 125.97 deg; joints [-10.503, -61.589, 110.858, 199.73, 34.406, -118.449, -235]
  MoveL 1538 to (81.34, -2.92, -143) mm, rotated rx -9.61 ry -16.54 rz 125.97 deg; joints [-10.598, -61.456, 110.812, 199.53, 34.467, -118.294, -235]
  MoveL 1539 to (80.83, -3.49, -143.95) mm, rotated rx -9.61 ry -16.54 rz 125.97 deg; joints [-10.637, -61.422, 110.823, 199.444, 34.502, -118.225, -235]
  MoveL 1540 to (80.18, -3.77, -144.72) mm, rotated rx -9.61 ry -16.54 rz 125.97 deg; joints [-10.67, -61.409, 110.857, 199.367, 34.538, -118.162, -235]
  MoveL 1541 to (79.8, -3.81, -145.04) mm, rotated rx -9.61 ry -16.54 rz 125.97 deg; joints [-10.685, -61.411, 110.882, 199.332, 34.557, -118.132, -235]
  MoveL 1542 to (79.39, -3.78, -145.31) mm, rotated rx -9.61 ry -16.54 rz 125.97 deg; joints [-10.698, -61.418, 110.913, 199.299, 34.577, -118.104, -235]
  MoveL 1543 to (78.47, -3.51, -145.74) mm, rotated rx -9.61 ry -16.54 rz 125.97 deg; joints [-10.719, -61.449, 110.992, 199.24, 34.619, -118.053, -235]
  MoveL 1544 to (77.42, -2.96, -146) mm, rotated rx -9.61 ry -16.54 rz 125.97 deg; joints [-10.735, -61.501, 111.094, 199.19, 34.662, -118.007, -235]
  MoveL 1545 to (76.23, -2.13, -146.08) mm, rotated rx -9.61 ry -16.54 rz 125.97 deg; joints [-10.745, -61.574, 111.219, 199.15, 34.709, -117.967, -235]
  MoveL 1546 to (75.81, -1.81, -146.08) mm, rotated rx -9.61 ry -16.54 rz 125.97 deg; joints [-10.747, -61.602, 111.263, 199.138, 34.724, -117.955, -235]
  MoveL 1547 to (75.49, -1.51, -146.03) mm, rotated rx -9.61 ry -16.54 rz 125.97 deg; joints [-10.747, -61.627, 111.301, 199.132, 34.736, -117.948, -235]
  MoveL 1548 to (75.17, -1.21, -145.97) mm, rotated rx -9.61 ry -16.54 rz 125.97 deg; joints [-10.746, -61.652, 111.337, 199.128, 34.747, -117.942, -235]
  MoveL 1549 to (74.81, -0.9, -145.93) mm, rotated rx -9.61 ry -16.54 rz 125.97 deg; joints [-10.747, -61.679, 111.378, 199.12, 34.76, -117.933, -235]
  MoveL 1550 to (74.43, -0.59, -145.92) mm, rotated rx -9.61 ry -16.54 rz 125.97 deg; joints [-10.748, -61.706, 111.42, 199.111, 34.774, -117.923, -235]
  MoveL 1551 to (74.01, -0.26, -145.91) mm, rotated rx -9.61 ry -16.54 rz 125.97 deg; joints [-10.75, -61.734, 111.466, 199.099, 34.79, -117.911, -235]
  MoveL 1552 to (73.59, 0.06, -145.91) mm, rotated rx -9.61 ry -16.54 rz 125.97 deg; joints [-10.753, -61.762, 111.51, 199.087, 34.805, -117.899, -235]
  MoveL 1553 to (73.18, 0.36, -145.93) mm, rotated rx -9.61 ry -16.54 rz 125.97 deg; joints [-10.756, -61.788, 111.554, 199.075, 34.821, -117.886, -235]
  MoveL 1554 to (72.78, 0.65, -145.94) mm, rotated rx -9.61 ry -16.54 rz 125.97 deg; joints [-10.758, -61.814, 111.596, 199.062, 34.836, -117.873, -235]
  MoveL 1555 to (72.42, 0.94, -145.92) mm, rotated rx -9.61 ry -16.54 rz 125.97 deg; joints [-10.76, -61.839, 111.636, 199.054, 34.849, -117.864, -235]
  MoveL 1556 to (72.07, 1.24, -145.88) mm, rotated rx -9.61 ry -16.54 rz 125.97 deg; joints [-10.76, -61.865, 111.675, 199.047, 34.862, -117.855, -235]
  MoveL 1557 to (71.66, 1.6, -145.83) mm, rotated rx -9.61 ry -16.54 rz 125.97 deg; joints [-10.76, -61.895, 111.722, 199.039, 34.877, -117.846, -235]
  MoveL 1558 to (71.13, 2.06, -145.77) mm, rotated rx -9.61 ry -16.54 rz 125.97 deg; joints [-10.761, -61.935, 111.781, 199.028, 34.896, -117.834, -235]
  MoveL 1559 to (70.63, 2.48, -145.75) mm, rotated rx -9.61 ry -16.54 rz 125.97 deg; joints [-10.763, -61.97, 111.836, 199.016, 34.914, -117.821, -235]
  MoveL 1560 to (68.56, 4.07, -145.75) mm, rotated rx -9.61 ry -16.54 rz 125.97 deg; joints [-10.775, -62.109, 112.059, 198.957, 34.991, -117.76, -235]
  MoveL 1561 to (68.07, 4.47, -145.71) mm, rotated rx -9.61 ry -16.54 rz 125.97 deg; joints [-10.776, -62.143, 112.112, 198.946, 35.008, -117.748, -235]
  MoveL 1562 to (67.65, 4.83, -145.65) mm, rotated rx -9.61 ry -16.54 rz 125.97 deg; joints [-10.776, -62.174, 112.159, 198.939, 35.024, -117.739, -235]
  MoveL 1563 to (67.49, 4.97, -145.51) mm, rotated rx -9.61 ry -16.54 rz 125.97 deg; joints [-10.771, -62.187, 112.178, 198.944, 35.031, -117.741, -235]
  MoveL 1564 to (67.59, 4.89, -145.24) mm, rotated rx -9.61 ry -16.54 rz 125.97 deg; joints [-10.76, -62.181, 112.17, 198.964, 35.031, -117.754, -235]
  MoveL 1565 to (67.93, 4.58, -144.84) mm, rotated rx -9.61 ry -16.54 rz 125.97 deg; joints [-10.741, -62.158, 112.136, 198.999, 35.025, -117.78, -235]
  MoveL 1566 to (68.27, 5.55, -144.03) mm, rotated rx -9.61 ry -16.54 rz 125.97 deg; joints [-10.709, -62.222, 112.153, 199.074, 34.987, -117.841, -235]
  MoveL 1567 to (67.69, 7.45, -143.82) mm, rotated rx -9.61 ry -16.54 rz 125.97 deg; joints [-10.707, -62.359, 112.27, 199.087, 34.969, -117.855, -235]
  MoveL 1568 to (67.08, 9.36, -143.66) mm, rotated rx -9.61 ry -16.54 rz 125.97 deg; joints [-10.707, -62.497, 112.39, 199.095, 34.951, -117.865, -235]
  MoveL 1569 to (66.45, 11.32, -143.5) mm, rotated rx -9.61 ry -16.54 rz 125.97 deg; joints [-10.708, -62.639, 112.512, 199.103, 34.933, -117.875, -235]
  MoveL 1570 to (65.89, 13.11, -143.21) mm, rotated rx -9.61 ry -16.54 rz 125.97 deg; joints [-10.702, -62.769, 112.625, 199.121, 34.917, -117.892, -235]
  MoveL 1571 to (65.24, 15.12, -143.02) mm, rotated rx -9.61 ry -16.54 rz 125.97 deg; joints [-10.701, -62.915, 112.75, 199.131, 34.898, -117.904, -235]
  MoveL 1572 to (64.56, 17.23, -142.84) mm, rotated rx -9.61 ry -16.54 rz 125.97 deg; joints [-10.701, -63.068, 112.882, 199.142, 34.877, -117.917, -235]
  MoveL 1573 to (63.86, 19.36, -142.75) mm, rotated rx -9.61 ry -16.54 rz 125.97 deg; joints [-10.705, -63.223, 113.014, 199.145, 34.856, -117.925, -235]
  MoveL 1574 to (63, 21.95, -142.66) mm, rotated rx -9.61 ry -16.54 rz 125.97 deg; joints [-10.711, -63.411, 113.175, 199.149, 34.829, -117.934, -235]
  MoveL 1575 to (62.38, 23.8, -142.56) mm, rotated rx -9.61 ry -16.54 rz 125.97 deg; joints [-10.713, -63.546, 113.292, 199.153, 34.811, -117.942, -235]
  MoveL 1576 to (61.8, 25.54, -142.34) mm, rotated rx -9.61 ry -16.54 rz 125.97 deg; joints [-10.711, -63.673, 113.401, 199.166, 34.795, -117.955, -235]
  MoveL 1577 to (61.16, 27.45, -142.15) mm, rotated rx -9.61 ry -16.54 rz 125.97 deg; joints [-10.71, -63.813, 113.521, 199.177, 34.776, -117.968, -235]
  MoveL 1578 to (60.47, 29.47, -142.03) mm, rotated rx -9.61 ry -16.54 rz 125.97 deg; joints [-10.712, -63.96, 113.647, 199.183, 34.755, -117.978, -235]
  MoveL 1579 to (59.79, 31.47, -141.85) mm, rotated rx -9.61 ry -16.54 rz 125.97 deg; joints [-10.712, -64.106, 113.772, 199.193, 34.736, -117.99, -235]
  MoveL 1580 to (59.11, 33.47, -141.73) mm, rotated rx -9.61 ry -16.54 rz 125.97 deg; joints [-10.715, -64.253, 113.897, 199.2, 34.715, -118, -235]
  MoveL 1581 to (58.4, 35.53, -141.55) mm, rotated rx -9.61 ry -16.54 rz 125.97 deg; joints [-10.715, -64.404, 114.026, 199.21, 34.694, -118.012, -235]
  MoveL 1582 to (57.7, 37.55, -141.43) mm, rotated rx -9.61 ry -16.54 rz 125.97 deg; joints [-10.717, -64.551, 114.152, 199.216, 34.673, -118.022, -235]
  MoveL 1583 to (56.99, 39.56, -141.2) mm, rotated rx -9.61 ry -16.54 rz 125.97 deg; joints [-10.715, -64.7, 114.279, 199.23, 34.653, -118.036, -235]
  MoveL 1584 to (56.29, 41.58, -141.09) mm, rotated rx -9.61 ry -16.54 rz 125.97 deg; joints [-10.718, -64.848, 114.405, 199.236, 34.631, -118.047, -235]
  MoveL 1585 to (55.59, 43.59, -140.97) mm, rotated rx -9.61 ry -16.54 rz 125.97 deg; joints [-10.721, -64.996, 114.53, 199.242, 34.609, -118.057, -235]
  MoveL 1586 to (54.86, 45.6, -140.75) mm, rotated rx -9.61 ry -16.54 rz 125.97 deg; joints [-10.719, -65.144, 114.657, 199.255, 34.59, -118.071, -235]
  MoveL 1587 to (54.16, 47.41, -140.55) mm, rotated rx -9.61 ry -16.54 rz 125.97 deg; joints [-10.717, -65.279, 114.776, 199.265, 34.575, -118.082, -235]
  MoveL 1588 to (53.46, 49.03, -140.26) mm, rotated rx -9.61 ry -16.54 rz 125.97 deg; joints [-10.712, -65.401, 114.888, 199.28, 34.567, -118.094, -235]
  MoveL 1589 to (52.73, 50.49, -139.85) mm, rotated rx -9.61 ry -16.54 rz 125.97 deg; joints [-10.701, -65.514, 114.997, 199.299, 34.566, -118.107, -235]
  MoveL 1590 to (52.69, 49, -138.92) mm, rotated rx -9.61 ry -16.54 rz 125.97 deg; joints [-10.658, -65.419, 114.96, 199.342, 34.629, -118.12, -235]
  MoveL 1591 to (52.62, 49.58, -138.91) mm, rotated rx -9.61 ry -16.54 rz 125.97 deg; joints [-10.659, -65.459, 114.984, 199.347, 34.615, -118.128, -235]
  MoveL 1592 to (52.59, 50.11, -138.89) mm, rotated rx -9.61 ry -16.54 rz 125.97 deg; joints [-10.66, -65.495, 115.005, 199.354, 34.599, -118.137, -235]
  MoveL 1593 to (52.61, 50.58, -138.83) mm, rotated rx -9.61 ry -16.54 rz 125.97 deg; joints [-10.658, -65.527, 115.02, 199.365, 34.584, -118.148, -235]
  MoveL 1594 to (52.65, 51.02, -138.76) mm, rotated rx -9.61 ry -16.54 rz 125.97 deg; joints [-10.656, -65.557, 115.032, 199.376, 34.568, -118.16, -235]
  MoveL 1595 to (52.73, 51.48, -138.71) mm, rotated rx -9.61 ry -16.54 rz 125.97 deg; joints [-10.655, -65.587, 115.042, 199.388, 34.549, -118.174, -235]
  MoveL 1596 to (52.83, 51.96, -138.68) mm, rotated rx -9.61 ry -16.54 rz 125.97 deg; joints [-10.654, -65.618, 115.05, 199.4, 34.527, -118.188, -235]
  MoveL 1597 to (52.96, 52.47, -138.66) mm, rotated rx -9.61 ry -16.54 rz 125.97 deg; joints [-10.654, -65.65, 115.057, 199.412, 34.503, -118.203, -235]
  MoveL 1598 to (53.1, 52.97, -138.66) mm, rotated rx -9.61 ry -16.54 rz 125.97 deg; joints [-10.655, -65.682, 115.063, 199.424, 34.479, -118.217, -235]
  MoveL 1599 to (53.21, 53.43, -138.65) mm, rotated rx -9.61 ry -16.54 rz 125.97 deg; joints [-10.655, -65.711, 115.07, 199.435, 34.458, -118.23, -235]
  MoveL 1600 to (53.3, 53.84, -138.63) mm, rotated rx -9.61 ry -16.54 rz 125.97 deg; joints [-10.655, -65.738, 115.077, 199.445, 34.439, -118.242, -235]
  MoveL 1601 to (53.41, 54.31, -138.61) mm, rotated rx -9.61 ry -16.54 rz 125.97 deg; joints [-10.655, -65.768, 115.083, 199.456, 34.417, -118.256, -235]
  MoveL 1602 to (53.55, 54.82, -138.61) mm, rotated rx -9.61 ry -16.54 rz 125.97 deg; joints [-10.656, -65.8, 115.089, 199.467, 34.393, -118.27, -235]
  MoveL 1603 to (53.7, 55.41, -138.59) mm, rotated rx -9.61 ry -16.54 rz 125.97 deg; joints [-10.656, -65.838, 115.097, 199.482, 34.365, -118.288, -235]
  MoveL 1604 to (53.86, 56.09, -138.55) mm, rotated rx -9.61 ry -16.54 rz 125.97 deg; joints [-10.655, -65.881, 115.108, 199.5, 34.334, -118.309, -235]
  MoveL 1605 to (54.01, 56.68, -138.53) mm, rotated rx -9.61 ry -16.54 rz 125.97 deg; joints [-10.655, -65.919, 115.116, 199.514, 34.306, -118.326, -235]
  MoveL 1606 to (54.16, 57.3, -138.51) mm, rotated rx -9.61 ry -16.54 rz 125.97 deg; joints [-10.655, -65.958, 115.125, 199.529, 34.277, -118.344, -235]
  MoveL 1607 to (54.31, 57.99, -138.47) mm, rotated rx -9.61 ry -16.54 rz 125.97 deg; joints [-10.654, -66.003, 115.136, 199.547, 34.245, -118.365, -235]
  MoveL 1608 to (54.46, 58.57, -138.45) mm, rotated rx -9.61 ry -16.54 rz 125.97 deg; joints [-10.654, -66.039, 115.143, 199.561, 34.218, -118.382, -235]
  MoveL 1609 to (54.6, 59.09, -138.45) mm, rotated rx -9.61 ry -16.54 rz 125.97 deg; joints [-10.655, -66.073, 115.15, 199.573, 34.192, -118.397, -235]
  MoveL 1610 to (55.01, 60.61, -138.45) mm, rotated rx -9.61 ry -16.54 rz 125.97 deg; joints [-10.657, -66.168, 115.167, 199.608, 34.118, -118.442, -235]
  MoveL 1611 to (55.46, 61.99, -138.54) mm, rotated rx -9.61 ry -16.54 rz 125.97 deg; joints [-10.662, -66.254, 115.176, 199.638, 34.045, -118.482, -235]
  MoveL 1612 to (55.97, 63.06, -138.79) mm, rotated rx -9.61 ry -16.54 rz 125.97 deg; joints [-10.673, -66.316, 115.169, 199.654, 33.977, -118.511, -235]
  MoveL 1613 to (56.54, 63.84, -139.21) mm, rotated rx -9.61 ry -16.54 rz 125.97 deg; joints [-10.691, -66.357, 115.145, 199.656, 33.913, -118.53, -235]
  MoveL 1614 to (56.84, 64.11, -139.48) mm, rotated rx -9.61 ry -16.54 rz 125.97 deg; joints [-10.702, -66.368, 115.127, 199.652, 33.883, -118.536, -235]
  MoveL 1615 to (57.16, 64.3, -139.8) mm, rotated rx -9.61 ry -16.54 rz 125.97 deg; joints [-10.715, -66.374, 115.105, 199.645, 33.853, -118.539, -235]
  MoveL 1616 to (57.85, 64.47, -140.56) mm, rotated rx -9.61 ry -16.54 rz 125.97 deg; joints [-10.745, -66.37, 115.05, 199.62, 33.799, -118.536, -235]
  MoveL 1617 to (58.6, 64.32, -141.49) mm, rotated rx -9.61 ry -16.54 rz 125.97 deg; joints [-10.781, -66.342, 114.977, 199.582, 33.749, -118.523, -235]
  MoveL 1618 to (60.27, 63.13, -143.85) mm, rotated rx -9.61 ry -16.54 rz 125.97 deg; joints [-10.871, -66.22, 114.784, 199.465, 33.662, -118.464, -235]
  MoveL 1619 to (61.69, 61.18, -146.21) mm, rotated rx -9.61 ry -16.54 rz 125.97 deg; joints [-10.961, -66.052, 114.587, 199.329, 33.614, -118.38, -235]
  MoveL 1620 to (62.35, 58.96, -147.9) mm, rotated rx -9.61 ry -16.54 rz 125.97 deg; joints [-11.024, -65.881, 114.445, 199.208, 33.628, -118.292, -235]
  MoveL 1621 to (62.4, 57.74, -148.49) mm, rotated rx -9.61 ry -16.54 rz 125.97 deg; joints [-11.045, -65.795, 114.396, 199.154, 33.658, -118.246, -235]
  MoveL 1622 to (62.26, 56.45, -148.91) mm, rotated rx -9.61 ry -16.54 rz 125.97 deg; joints [-11.06, -65.708, 114.36, 199.103, 33.703, -118.199, -235]
  MoveL 1623 to (61.41, 53.66, -149.25) mm, rotated rx -9.61 ry -16.54 rz 125.97 deg; joints [-11.071, -65.533, 114.331, 199.014, 33.839, -118.101, -235]
  MoveL 1624 to (59.8, 49.79, -149.25) mm, rotated rx -9.61 ry -16.54 rz 125.97 deg; joints [-11.068, -65.3, 114.329, 198.907, 34.059, -117.97, -235]
  MoveL 1625 to (59.6, 49.28, -149.27) mm, rotated rx -9.61 ry -16.54 rz 125.97 deg; joints [-11.068, -65.268, 114.327, 198.893, 34.086, -117.952, -235]
  MoveL 1626 to (59.43, 48.78, -149.31) mm, rotated rx -9.61 ry -16.54 rz 125.97 deg; joints [-11.069, -65.238, 114.324, 198.878, 34.112, -117.935, -235]
  MoveL 1627 to (59.26, 48.28, -149.37) mm, rotated rx -9.61 ry -16.54 rz 125.97 deg; joints [-11.071, -65.206, 114.319, 198.861, 34.137, -117.918, -235]
  MoveL 1628 to (59.12, 47.78, -149.45) mm, rotated rx -9.61 ry -16.54 rz 125.97 deg; joints [-11.074, -65.174, 114.313, 198.845, 34.161, -117.9, -235]
  MoveL 1629 to (58.98, 47.29, -149.53) mm, rotated rx -9.61 ry -16.54 rz 125.97 deg; joints [-11.076, -65.143, 114.307, 198.828, 34.184, -117.883, -235]
  MoveL 1630 to (58.82, 46.84, -149.57) mm, rotated rx -9.61 ry -16.54 rz 125.97 deg; joints [-11.078, -65.115, 114.304, 198.815, 34.208, -117.867, -235]
  MoveL 1631 to (58.64, 46.39, -149.59) mm, rotated rx -9.61 ry -16.54 rz 125.97 deg; joints [-11.078, -65.087, 114.303, 198.802, 34.232, -117.852, -235]
  MoveL 1632 to (58.44, 45.91, -149.59) mm, rotated rx -9.61 ry -16.54 rz 125.97 deg; joints [-11.077, -65.058, 114.302, 198.789, 34.259, -117.836, -235]
  MoveL 1633 to (58.22, 45.32, -149.62) mm, rotated rx -9.61 ry -16.54 rz 125.97 deg; joints [-11.078, -65.022, 114.299, 198.772, 34.291, -117.816, -235]
  MoveL 1634 to (57.99, 44.68, -149.68) mm, rotated rx -9.61 ry -16.54 rz 125.97 deg; joints [-11.08, -64.982, 114.295, 198.752, 34.324, -117.793, -235]
  MoveL 1635 to (57.8, 44.11, -149.7) mm, rotated rx -9.61 ry -16.54 rz 125.97 deg; joints [-11.08, -64.947, 114.291, 198.737, 34.353, -117.776, -235]
  MoveL 1636 to (57.66, 43.58, -149.71) mm, rotated rx -9.61 ry -16.54 rz 125.97 deg; joints [-11.08, -64.913, 114.283, 198.725, 34.379, -117.761, -235]
  MoveL 1637 to (57.56, 43.03, -149.71) mm, rotated rx -9.61 ry -16.54 rz 125.97 deg; joints [-11.079, -64.878, 114.272, 198.716, 34.401, -117.748, -235]
  MoveL 1638 to (57.59, 42.45, -149.71) mm, rotated rx -9.61 ry -16.54 rz 125.97 deg; joints [-11.077, -64.839, 114.251, 198.71, 34.419, -117.74, -235]
  MoveL 1639 to (57.68, 41.85, -149.71) mm, rotated rx -9.61 ry -16.54 rz 125.97 deg; joints [-11.076, -64.796, 114.223, 198.706, 34.433, -117.734, -235]
  MoveL 1640 to (57.8, 43.42, -150.67) mm, rotated rx -9.61 ry -16.54 rz 125.97 deg; joints [-11.119, -64.895, 114.258, 198.663, 34.363, -117.722, -235]
  MoveL 1641 to (58.26, 42.26, -151.09) mm, rotated rx -9.61 ry -16.54 rz 125.97 deg; joints [-11.132, -64.807, 114.177, 198.638, 34.368, -117.704, -235]
  MoveL 1642 to (58.69, 40.91, -151.42) mm, rotated rx -9.61 ry -16.54 rz 125.97 deg; joints [-11.141, -64.707, 114.094, 198.617, 34.382, -117.685, -235]
  MoveL 1643 to (59.1, 39.36, -151.67) mm, rotated rx -9.61 ry -16.54 rz 125.97 deg; joints [-11.145, -64.595, 114.006, 198.597, 34.404, -117.666, -235]
  MoveL 1644 to (59.54, 37.27, -151.78) mm, rotated rx -9.61 ry -16.54 rz 125.97 deg; joints [-11.143, -64.446, 113.898, 198.583, 34.443, -117.646, -235]
  MoveL 1645 to (60, 35.19, -152.01) mm, rotated rx -9.61 ry -16.54 rz 125.97 deg; joints [-11.145, -64.298, 113.788, 198.561, 34.479, -117.622, -235]
  MoveL 1646 to (60.43, 33.1, -152.13) mm, rotated rx -9.61 ry -16.54 rz 125.97 deg; joints [-11.143, -64.15, 113.68, 198.546, 34.517, -117.602, -235]
  MoveL 1647 to (60.86, 31.01, -152.24) mm, rotated rx -9.61 ry -16.54 rz 125.97 deg; joints [-11.141, -64.002, 113.572, 198.531, 34.556, -117.582, -235]
  MoveL 1648 to (61.3, 28.93, -152.48) mm, rotated rx -9.61 ry -16.54 rz 125.97 deg; joints [-11.143, -63.853, 113.462, 198.509, 34.592, -117.557, -235]
  MoveL 1649 to (61.73, 26.84, -152.6) mm, rotated rx -9.61 ry -16.54 rz 125.97 deg; joints [-11.141, -63.705, 113.354, 198.495, 34.63, -117.538, -235]
  MoveL 1650 to (62.15, 24.75, -152.72) mm, rotated rx -9.61 ry -16.54 rz 125.97 deg; joints [-11.139, -63.557, 113.245, 198.48, 34.667, -117.518, -235]
  MoveL 1651 to (62.64, 22.34, -152.88) mm, rotated rx -9.61 ry -16.54 rz 125.97 deg; joints [-11.137, -63.387, 113.119, 198.462, 34.71, -117.495, -235]
  MoveL 1652 to (63.05, 20.28, -153.07) mm, rotated rx -9.61 ry -16.54 rz 125.97 deg; joints [-11.139, -63.241, 113.011, 198.443, 34.746, -117.472, -235]
  MoveL 1653 to (63.5, 18.01, -153.27) mm, rotated rx -9.61 ry -16.54 rz 125.97 deg; joints [-11.139, -63.081, 112.893, 198.423, 34.785, -117.449, -235]
  MoveL 1654 to (63.93, 15.79, -153.52) mm, rotated rx -9.61 ry -16.54 rz 125.97 deg; joints [-11.142, -62.924, 112.776, 198.4, 34.823, -117.423, -235]
  MoveL 1655 to (64.34, 13.7, -153.64) mm, rotated rx -9.61 ry -16.54 rz 125.97 deg; joints [-11.14, -62.776, 112.667, 198.385, 34.86, -117.404, -235]
  MoveL 1656 to (64.76, 11.61, -153.64) mm, rotated rx -9.61 ry -16.54 rz 125.97 deg; joints [-11.133, -62.629, 112.558, 198.38, 34.897, -117.39, -235]
  MoveL 1657 to (65.16, 9.54, -153.72) mm, rotated rx -9.61 ry -16.54 rz 125.97 deg; joints [-11.13, -62.484, 112.45, 198.369, 34.933, -117.374, -235]
  MoveL 1658 to (65.53, 7.51, -153.93) mm, rotated rx -9.61 ry -16.54 rz 125.97 deg; joints [-11.132, -62.341, 112.345, 198.349, 34.968, -117.351, -235]
  MoveL 1659 to (65.92, 5.25, -154.28) mm, rotated rx -9.61 ry -16.54 rz 125.97 deg; joints [-11.139, -62.181, 112.226, 198.318, 35.006, -117.321, -235]
  MoveL 1660 to (66.23, 3.47, -154.5) mm, rotated rx -9.61 ry -16.54 rz 125.97 deg; joints [-11.142, -62.056, 112.134, 198.299, 35.037, -117.3, -235]
  MoveL 1661 to (66.63, 1.04, -154.79) mm, rotated rx -9.61 ry -16.54 rz 125.97 deg; joints [-11.146, -61.886, 112.01, 198.271, 35.079, -117.27, -235]
  MoveL 1662 to (67.03, -1.13, -154.9) mm, rotated rx -9.61 ry -16.54 rz 125.97 deg; joints [-11.144, -61.734, 111.896, 198.258, 35.116, -117.252, -235]
  MoveL 1663 to (67.44, -3.22, -154.91) mm, rotated rx -9.61 ry -16.54 rz 125.97 deg; joints [-11.137, -61.588, 111.785, 198.253, 35.151, -117.239, -235]
  MoveL 1664 to (67.1, -4.04, -155.7) mm, rotated rx -9.61 ry -16.54 rz 125.97 deg; joints [-11.169, -61.534, 111.773, 198.182, 35.185, -117.183, -235]
  MoveL 1665 to (66.85, -3.68, -156.09) mm, rotated rx -9.61 ry -16.54 rz 125.97 deg; joints [-11.187, -61.56, 111.803, 198.152, 35.185, -117.162, -235]
  MoveL 1666 to (66.78, -3.55, -156.34) mm, rotated rx -9.61 ry -16.54 rz 125.97 deg; joints [-11.198, -61.567, 111.81, 198.134, 35.183, -117.151, -235]
  MoveL 1667 to (66.88, -3.66, -156.46) mm, rotated rx -9.61 ry -16.54 rz 125.97 deg; joints [-11.202, -61.558, 111.797, 198.129, 35.178, -117.149, -235]
  MoveL 1668 to (67.14, -3.95, -156.48) mm, rotated rx -9.61 ry -16.54 rz 125.97 deg; joints [-11.201, -61.535, 111.765, 198.134, 35.17, -117.154, -235]
  MoveL 1669 to (67.47, -4.28, -156.49) mm, rotated rx -9.61 ry -16.54 rz 125.97 deg; joints [-11.199, -61.507, 111.727, 198.142, 35.16, -117.162, -235]
  MoveL 1670 to (68.58, -5.39, -156.49) mm, rotated rx -9.61 ry -16.54 rz 125.97 deg; joints [-11.192, -61.416, 111.597, 198.171, 35.125, -117.191, -235]
  MoveL 1671 to (68.96, -5.79, -156.51) mm, rotated rx -9.61 ry -16.54 rz 125.97 deg; joints [-11.19, -61.384, 111.552, 198.18, 35.113, -117.199, -235]
  MoveL 1672 to (69.33, -6.21, -156.56) mm, rotated rx -9.61 ry -16.54 rz 125.97 deg; joints [-11.189, -61.35, 111.507, 198.186, 35.102, -117.206, -235]
  MoveL 1673 to (69.7, -6.65, -156.64) mm, rotated rx -9.61 ry -16.54 rz 125.97 deg; joints [-11.19, -61.315, 111.461, 198.19, 35.092, -117.211, -235]
  MoveL 1674 to (70.06, -7.06, -156.7) mm, rotated rx -9.61 ry -16.54 rz 125.97 deg; joints [-11.19, -61.281, 111.416, 198.195, 35.081, -117.218, -235]
  MoveL 1675 to (70.42, -7.45, -156.72) mm, rotated rx -9.61 ry -16.54 rz 125.97 deg; joints [-11.189, -61.25, 111.372, 198.202, 35.07, -117.226, -235]
  MoveL 1676 to (70.76, -7.81, -156.74) mm, rotated rx -9.61 ry -16.54 rz 125.97 deg; joints [-11.187, -61.22, 111.331, 198.21, 35.059, -117.234, -235]
  MoveL 1677 to (71.06, -8.16, -156.79) mm, rotated rx -9.61 ry -16.54 rz 125.97 deg; joints [-11.187, -61.192, 111.294, 198.215, 35.05, -117.239, -235]
  MoveL 1678 to (71.36, -8.49, -156.83) mm, rotated rx -9.61 ry -16.54 rz 125.97 deg; joints [-11.186, -61.166, 111.258, 198.219, 35.042, -117.244, -235]
  MoveL 1679 to (71.7, -8.85, -156.84) mm, rotated rx -9.61 ry -16.54 rz 125.97 deg; joints [-11.185, -61.136, 111.217, 198.227, 35.031, -117.253, -235]
  MoveL 1680 to (72.1, -9.27, -156.86) mm, rotated rx -9.61 ry -16.54 rz 125.97 deg; joints [-11.183, -61.102, 111.169, 198.237, 35.018, -117.262, -235]
  MoveL 1681 to (72.57, -9.8, -156.91) mm, rotated rx -9.61 ry -16.54 rz 125.97 deg; joints [-11.182, -61.059, 111.112, 198.245, 35.004, -117.271, -235]
  MoveL 1682 to (72.98, -10.24, -156.94) mm, rotated rx -9.61 ry -16.54 rz 125.97 deg; joints [-11.18, -61.023, 111.062, 198.254, 34.992, -117.281, -235]
  MoveL 1683 to (74.47, -11.73, -156.95) mm, rotated rx -9.61 ry -16.54 rz 125.97 deg; joints [-11.171, -60.902, 110.888, 198.293, 34.944, -117.319, -235]
  MoveL 1684 to (76.32, -13.98, -157.27) mm, rotated rx -9.61 ry -16.54 rz 125.97 deg; joints [-11.171, -60.721, 110.652, 198.317, 34.891, -117.349, -235]
  MoveL 1685 to (76.94, -15.12, -157.69) mm, rotated rx -9.61 ry -16.54 rz 125.97 deg; joints [-11.182, -60.634, 110.555, 198.303, 34.88, -117.343, -235]
  MoveL 1686 to (77.36, -16.25, -158.26) mm, rotated rx -9.61 ry -16.54 rz 125.97 deg; joints [-11.201, -60.549, 110.472, 198.271, 34.878, -117.321, -235]
  MoveL 1687 to (77.61, -18.55, -159.91) mm, rotated rx -9.61 ry -16.54 rz 125.97 deg; joints [-11.261, -60.383, 110.347, 198.155, 34.905, -117.235, -235]
  MoveL 1688 to (77.06, -20.86, -162.22) mm, rotated rx -9.61 ry -16.54 rz 125.97 deg; joints [-11.35, -60.224, 110.277, 197.969, 34.971, -117.092, -235]
  MoveL 1689 to (75.98, -22.58, -164.53) mm, rotated rx -9.61 ry -16.54 rz 125.97 deg; joints [-11.443, -60.112, 110.27, 197.77, 35.053, -116.936, -235]
  MoveL 1690 to (75.35, -22.98, -165.43) mm, rotated rx -9.61 ry -16.54 rz 125.97 deg; joints [-11.482, -60.089, 110.295, 197.687, 35.091, -116.871, -235]
  MoveL 1691 to (74.66, -23.09, -166.17) mm, rotated rx -9.61 ry -16.54 rz 125.97 deg; joints [-11.514, -60.089, 110.337, 197.615, 35.126, -116.813, -235]
  MoveL 1692 to (74.29, -23.02, -166.48) mm, rotated rx -9.61 ry -16.54 rz 125.97 deg; joints [-11.528, -60.096, 110.365, 197.583, 35.143, -116.788, -235]
  MoveL 1693 to (73.91, -22.89, -166.75) mm, rotated rx -9.61 ry -16.54 rz 125.97 deg; joints [-11.541, -60.11, 110.398, 197.554, 35.159, -116.764, -235]
  MoveL 1694 to (73.09, -22.39, -167.16) mm, rotated rx -9.61 ry -16.54 rz 125.97 deg; joints [-11.562, -60.153, 110.478, 197.503, 35.189, -116.722, -235]
  MoveL 1695 to (72.21, -21.58, -167.41) mm, rotated rx -9.61 ry -16.54 rz 125.97 deg; joints [-11.578, -60.218, 110.576, 197.463, 35.218, -116.688, -235]
  MoveL 1696 to (71.28, -20.48, -167.49) mm, rotated rx -9.61 ry -16.54 rz 125.97 deg; joints [-11.589, -60.305, 110.692, 197.434, 35.243, -116.662, -235]
  MoveL 1697 to (69.04, -17.57, -167.49) mm, rotated rx -9.61 ry -16.54 rz 125.97 deg; joints [-11.606, -60.531, 110.98, 197.38, 35.299, -116.612, -235]
  MoveL 1698 to (68.76, -17.2, -167.48) mm, rotated rx -9.61 ry -16.54 rz 125.97 deg; joints [-11.607, -60.56, 111.017, 197.374, 35.306, -116.607, -235]
  MoveL 1699 to (68.53, -16.87, -167.45) mm, rotated rx -9.61 ry -16.54 rz 125.97 deg; joints [-11.608, -60.586, 111.048, 197.371, 35.311, -116.603, -235]
  MoveL 1700 to (68.25, -16.48, -167.43) mm, rotated rx -9.61 ry -16.54 rz 125.97 deg; joints [-11.61, -60.616, 111.085, 197.365, 35.318, -116.597, -235]
  MoveL 1701 to (66.01, -13.58, -167.43) mm, rotated rx -9.61 ry -16.54 rz 125.97 deg; joints [-11.627, -60.843, 111.373, 197.311, 35.373, -116.548, -235]
  MoveL 1702 to (65.69, -13.14, -167.41) mm, rotated rx -9.61 ry -16.54 rz 125.97 deg; joints [-11.629, -60.877, 111.415, 197.305, 35.379, -116.542, -235]
  MoveL 1703 to (65.4, -12.68, -167.38) mm, rotated rx -9.61 ry -16.54 rz 125.97 deg; joints [-11.63, -60.912, 111.456, 197.301, 35.385, -116.538, -235]
  MoveL 1704 to (65.19, -12.24, -167.33) mm, rotated rx -9.61 ry -16.54 rz 125.97 deg; joints [-11.63, -60.945, 111.49, 197.3, 35.386, -116.537, -235]
  MoveL 1705 to (65.05, -11.88, -167.27) mm, rotated rx -9.61 ry -16.54 rz 125.97 deg; joints [-11.629, -60.972, 111.515, 197.302, 35.385, -116.539, -235]
  MoveL 1706 to (65.01, -11.69, -167.1) mm, rotated rx -9.61 ry -16.54 rz 125.97 deg; joints [-11.623, -60.986, 111.527, 197.313, 35.384, -116.546, -235]
  MoveL 1707 to (65.04, -11.67, -166.77) mm, rotated rx -9.61 ry -16.54 rz 125.97 deg; joints [-11.61, -60.989, 111.53, 197.335, 35.386, -116.561, -235]
  MoveL 1708 to (65.12, -11.8, -166.26) mm, rotated rx -9.61 ry -16.54 rz 125.97 deg; joints [-11.588, -60.982, 111.524, 197.37, 35.391, -116.583, -235]
  MoveL 1709 to (65.63, -11.15, -164.8) mm, rotated rx -9.61 ry -16.54 rz 125.97 deg; joints [-11.528, -61.027, 111.524, 197.486, 35.36, -116.669, -235]
  MoveL 1710 to (65.35, -6.89, -164.8) mm, rotated rx -9.61 ry -16.54 rz 125.97 deg; joints [-11.541, -61.316, 111.708, 197.51, 35.258, -116.71, -235]
  MoveL 1711 to (65.22, -4.86, -164.75) mm, rotated rx -9.61 ry -16.54 rz 125.97 deg; joints [-11.545, -61.455, 111.796, 197.525, 35.208, -116.732, -235]
  MoveL 1712 to (65.1, -2.88, -164.67) mm, rotated rx -9.61 ry -16.54 rz 125.97 deg; joints [-11.547, -61.589, 111.881, 197.542, 35.161, -116.756, -235]
  MoveL 1713 to (64.97, -0.87, -164.58) mm, rotated rx -9.61 ry -16.54 rz 125.97 deg; joints [-11.55, -61.726, 111.968, 197.56, 35.112, -116.78, -235]
  MoveL 1714 to (64.84, 1.09, -164.48) mm, rotated rx -9.61 ry -16.54 rz 125.97 deg; joints [-11.551, -61.86, 112.052, 197.579, 35.064, -116.804, -235]
  MoveL 1715 to (64.73, 3.19, -164.44) mm, rotated rx -9.61 ry -16.54 rz 125.97 deg; joints [-11.556, -62.003, 112.139, 197.595, 35.011, -116.828, -235]
  MoveL 1716 to (64.69, 5.39, -164.41) mm, rotated rx -9.61 ry -16.54 rz 125.97 deg; joints [-11.561, -62.151, 112.224, 197.615, 34.95, -116.856, -235]
  MoveL 1717 to (64.43, 7.87, -164.24) mm, rotated rx -9.61 ry -16.54 rz 125.97 deg; joints [-11.562, -62.322, 112.338, 197.638, 34.894, -116.886, -235]
  MoveL 1718 to (64.28, 10.11, -163.99) mm, rotated rx -9.61 ry -16.54 rz 125.97 deg; joints [-11.558, -62.476, 112.434, 197.669, 34.841, -116.92, -235]
  MoveL 1719 to (64.14, 12.3, -163.86) mm, rotated rx -9.61 ry -16.54 rz 125.97 deg; joints [-11.559, -62.626, 112.527, 197.692, 34.786, -116.949, -235]
  MoveL 1720 to (63.99, 14.43, -163.62) mm, rotated rx -9.61 ry -16.54 rz 125.97 deg; joints [-11.556, -62.772, 112.619, 197.722, 34.734, -116.982, -235]
  MoveL 1721 to (63.84, 16.56, -163.5) mm, rotated rx -9.61 ry -16.54 rz 125.97 deg; joints [-11.557, -62.918, 112.708, 197.744, 34.681, -117.011, -235]
  MoveL 1722 to (63.69, 18.69, -163.38) mm, rotated rx -9.61 ry -16.54 rz 125.97 deg; joints [-11.559, -63.064, 112.798, 197.766, 34.627, -117.039, -235]
  MoveL 1723 to (63.53, 20.82, -163.14) mm, rotated rx -9.61 ry -16.54 rz 125.97 deg; joints [-11.555, -63.211, 112.89, 197.796, 34.575, -117.072, -235]
  MoveL 1724 to (63.37, 22.94, -163.02) mm, rotated rx -9.61 ry -16.54 rz 125.97 deg; joints [-11.557, -63.357, 112.98, 197.819, 34.521, -117.101, -235]
  MoveL 1725 to (63.21, 25.07, -162.9) mm, rotated rx -9.61 ry -16.54 rz 125.97 deg; joints [-11.558, -63.503, 113.069, 197.841, 34.467, -117.13, -235]
  MoveL 1726 to (63.05, 27.2, -162.79) mm, rotated rx -9.61 ry -16.54 rz 125.97 deg; joints [-11.56, -63.649, 113.158, 197.864, 34.413, -117.159, -235]
  MoveL 1727 to (62.86, 29.32, -162.56) mm, rotated rx -9.61 ry -16.54 rz 125.97 deg; joints [-11.557, -63.796, 113.25, 197.893, 34.361, -117.192, -235]
  MoveL 1728 to (62.7, 31.45, -162.45) mm, rotated rx -9.61 ry -16.54 rz 125.97 deg; joints [-11.559, -63.942, 113.339, 197.916, 34.306, -117.221, -235]
  MoveL 1729 to (62.51, 33.23, -162.19) mm, rotated rx -9.61 ry -16.54 rz 125.97 deg; joints [-11.554, -64.066, 113.418, 197.944, 34.264, -117.251, -235]
  MoveL 1730 to (62.33, 34.87, -161.87) mm, rotated rx -9.61 ry -16.54 rz 125.97 deg; joints [-11.546, -64.181, 113.493, 197.976, 34.228, -117.282, -235]
  MoveL 1731 to (62.12, 36.43, -161.45) mm, rotated rx -9.61 ry -16.54 rz 125.97 deg; joints [-11.534, -64.291, 113.568, 198.013, 34.196, -117.315, -235]
  MoveL 1732 to (61.52, 34.8, -160.5) mm, rotated rx -9.61 ry -16.54 rz 125.97 deg; joints [-11.492, -64.197, 113.569, 198.039, 34.295, -117.309, -235]
  MoveL 1733 to (61.52, 35.43, -160.37) mm, rotated rx -9.61 ry -16.54 rz 125.97 deg; joints [-11.488, -64.241, 113.592, 198.054, 34.277, -117.324, -235]
  MoveL 1734 to (61.58, 36.01, -160.28) mm, rotated rx -9.61 ry -16.54 rz 125.97 deg; joints [-11.486, -64.279, 113.608, 198.068, 34.256, -117.339, -235]
  MoveL 1735 to (61.75, 36.53, -160.25) mm, rotated rx -9.61 ry -16.54 rz 125.97 deg; joints [-11.485, -64.311, 113.613, 198.082, 34.23, -117.355, -235]
  MoveL 1736 to (61.96, 37.02, -160.23) mm, rotated rx -9.61 ry -16.54 rz 125.97 deg; joints [-11.485, -64.341, 113.613, 198.096, 34.202, -117.371, -235]
  MoveL 1737 to (63.78, 40.22, -160.22) mm, rotated rx -9.61 ry -16.54 rz 125.97 deg; joints [-11.486, -64.526, 113.58, 198.195, 33.995, -117.492, -235]
  MoveL 1738 to (64, 40.62, -160.21) mm, rotated rx -9.61 ry -16.54 rz 125.97 deg; joints [-11.485, -64.55, 113.576, 198.209, 33.969, -117.507, -235]
  MoveL 1739 to (64.2, 41, -160.18) mm, rotated rx -9.61 ry -16.54 rz 125.97 deg; joints [-11.484, -64.572, 113.574, 198.222, 33.946, -117.522, -235]
  MoveL 1740 to (64.43, 41.42, -160.17) mm, rotated rx -9.61 ry -16.54 rz 125.97 deg; joints [-11.484, -64.596, 113.57, 198.235, 33.919, -117.538, -235]
  MoveL 1741 to (64.69, 41.87, -160.17) mm, rotated rx -9.61 ry -16.54 rz 125.97 deg; joints [-11.484, -64.622, 113.565, 198.25, 33.889, -117.556, -235]
  MoveL 1742 to (65.48, 43.23, -160.17) mm, rotated rx -9.61 ry -16.54 rz 125.97 deg; joints [-11.484, -64.701, 113.549, 198.293, 33.8, -117.608, -235]
  MoveL 1743 to (65.78, 43.78, -160.15) mm, rotated rx -9.61 ry -16.54 rz 125.97 deg; joints [-11.484, -64.732, 113.544, 198.312, 33.765, -117.63, -235]
  MoveL 1744 to (66.11, 44.42, -160.12) mm, rotated rx -9.61 ry -16.54 rz 125.97 deg; joints [-11.482, -64.77, 113.54, 198.333, 33.726, -117.655, -235]
  MoveL 1745 to (66.42, 44.98, -160.09) mm, rotated rx -9.61 ry -16.54 rz 125.97 deg; joints [-11.482, -64.802, 113.535, 198.352, 33.69, -117.677, -235]
  MoveL 1746 to (66.94, 45.89, -160.09) mm, rotated rx -9.61 ry -16.54 rz 125.97 deg; joints [-11.482, -64.854, 113.524, 198.382, 33.631, -117.713, -235]
  MoveL 1747 to (67.73, 47.11, -160.18) mm, rotated rx -9.61 ry -16.54 rz 125.97 deg; joints [-11.485, -64.922, 113.502, 198.418, 33.545, -117.76, -235]
  MoveL 1748 to (68.49, 48.02, -160.43) mm, rotated rx -9.61 ry -16.54 rz 125.97 deg; joints [-11.495, -64.968, 113.47, 198.44, 33.468, -117.794, -235]
  MoveL 1749 to (69.23, 48.61, -160.85) mm, rotated rx -9.61 ry -16.54 rz 125.97 deg; joints [-11.511, -64.993, 113.426, 198.445, 33.4, -117.815, -235]
  MoveL 1750 to (69.6, 48.79, -161.12) mm, rotated rx -9.61 ry -16.54 rz 125.97 deg; joints [-11.521, -64.997, 113.401, 198.442, 33.37, -117.82, -235]
  MoveL 1751 to (69.96, 48.9, -161.44) mm, rotated rx -9.61 ry -16.54 rz 125.97 deg; joints [-11.533, -64.996, 113.372, 198.435, 33.341, -117.822, -235]
  MoveL 1752 to (70.66, 48.87, -162.19) mm, rotated rx -9.61 ry -16.54 rz 125.97 deg; joints [-11.562, -64.977, 113.308, 198.408, 33.292, -117.816, -235]
  MoveL 1753 to (71.34, 48.53, -163.12) mm, rotated rx -9.61 ry -16.54 rz 125.97 deg; joints [-11.596, -64.937, 113.232, 198.366, 33.251, -117.796, -235]
  MoveL 1754 to (72.65, 46.92, -165.47) mm, rotated rx -9.61 ry -16.54 rz 125.97 deg; joints [-11.684, -64.792, 113.049, 198.234, 33.197, -117.717, -235]
  MoveL 1755 to (73.51, 44.65, -167.82) mm, rotated rx -9.61 ry -16.54 rz 125.97 deg; joints [-11.771, -64.611, 112.879, 198.079, 33.188, -117.61, -235]
  MoveL 1756 to (73.58, 42.31, -169.5) mm, rotated rx -9.61 ry -16.54 rz 125.97 deg; joints [-11.834, -64.443, 112.776, 197.941, 33.237, -117.501, -235]
  MoveL 1757 to (73.31, 41.11, -170.09) mm, rotated rx -9.61 ry -16.54 rz 125.97 deg; joints [-11.856, -64.364, 112.75, 197.878, 33.283, -117.445, -235]
  MoveL 1758 to (72.85, 39.89, -170.51) mm, rotated rx -9.61 ry -16.54 rz 125.97 deg; joints [-11.872, -64.288, 112.741, 197.82, 33.343, -117.39, -235]
  MoveL 1759 to (71.32, 37.41, -170.85) mm, rotated rx -9.61 ry -16.54 rz 125.97 deg; joints [-11.886, -64.146, 112.773, 197.716, 33.507, -117.277, -235]
  MoveL 1760 to (69.41, 34.91, -170.85) mm, rotated rx -9.61 ry -16.54 rz 125.97 deg; joints [-11.888, -64.011, 112.838, 197.622, 33.697, -117.166, -235]
  MoveL 1761 to (68.85, 34.1, -170.89) mm, rotated rx -9.61 ry -16.54 rz 125.97 deg; joints [-11.89, -63.966, 112.854, 197.591, 33.755, -117.131, -235]
  MoveL 1762 to (68.53, 33.69, -170.89) mm, rotated rx -9.61 ry -16.54 rz 125.97 deg; joints [-11.89, -63.944, 112.864, 197.575, 33.786, -117.112, -235]
  MoveL 1763 to (68.21, 33.26, -170.9) mm, rotated rx -9.61 ry -16.54 rz 125.97 deg; joints [-11.89, -63.92, 112.875, 197.559, 33.819, -117.093, -235]
  MoveL 1764 to (67.87, 32.8, -170.92) mm, rotated rx -9.61 ry -16.54 rz 125.97 deg; joints [-11.892, -63.895, 112.885, 197.541, 33.852, -117.073, -235]
  MoveL 1765 to (67.51, 32.26, -170.98) mm, rotated rx -9.61 ry -16.54 rz 125.97 deg; joints [-11.894, -63.865, 112.895, 197.519, 33.89, -117.048, -235]
  MoveL 1766 to (67.18, 31.79, -171.01) mm, rotated rx -9.61 ry -16.54 rz 125.97 deg; joints [-11.896, -63.838, 112.905, 197.501, 33.924, -117.027, -235]
  MoveL 1767 to (66.87, 31.36, -171.02) mm, rotated rx -9.61 ry -16.54 rz 125.97 deg; joints [-11.896, -63.815, 112.914, 197.485, 33.955, -117.009, -235]
  MoveL 1768 to (66.59, 30.97, -171.05) mm, rotated rx -9.61 ry -16.54 rz 125.97 deg; joints [-11.898, -63.793, 112.922, 197.469, 33.983, -116.991, -235]
  MoveL 1769 to (66.35, 30.59, -171.1) mm, rotated rx -9.61 ry -16.54 rz 125.97 deg; joints [-11.9, -63.771, 112.927, 197.453, 34.009, -116.974, -235]
  MoveL 1770 to (66.09, 30.21, -171.14) mm, rotated rx -9.61 ry -16.54 rz 125.97 deg; joints [-11.901, -63.75, 112.934, 197.438, 34.035, -116.958, -235]
  MoveL 1771 to (65.79, 29.8, -171.15) mm, rotated rx -9.61 ry -16.54 rz 125.97 deg; joints [-11.902, -63.727, 112.943, 197.423, 34.066, -116.94, -235]
  MoveL 1772 to (65.49, 29.38, -171.16) mm, rotated rx -9.61 ry -16.54 rz 125.97 deg; joints [-11.902, -63.704, 112.952, 197.408, 34.096, -116.922, -235]
  MoveL 1773 to (65.2, 28.95, -171.17) mm, rotated rx -9.61 ry -16.54 rz 125.97 deg; joints [-11.903, -63.68, 112.959, 197.394, 34.126, -116.905, -235]
  MoveL 1774 to (64.98, 28.52, -171.18) mm, rotated rx -9.61 ry -16.54 rz 125.97 deg; joints [-11.903, -63.654, 112.961, 197.38, 34.153, -116.889, -235]
  MoveL 1775 to (64.82, 28.07, -171.22) mm, rotated rx -9.61 ry -16.54 rz 125.97 deg; joints [-11.904, -63.626, 112.958, 197.368, 34.176, -116.876, -235]
  MoveL 1776 to (64.72, 27.63, -171.26) mm, rotated rx -9.61 ry -16.54 rz 125.97 deg; joints [-11.905, -63.598, 112.949, 197.358, 34.194, -116.864, -235]
  MoveL 1777 to (64.66, 27.17, -171.31) mm, rotated rx -9.61 ry -16.54 rz 125.97 deg; joints [-11.906, -63.568, 112.938, 197.349, 34.212, -116.853, -235]
  MoveL 1778 to (65.12, 28.63, -172.27) mm, rotated rx -9.61 ry -16.54 rz 125.97 deg; joints [-11.948, -63.652, 112.942, 197.313, 34.127, -116.849, -235]
  MoveL 1779 to (65.18, 26.91, -172.65) mm, rotated rx -9.61 ry -16.54 rz 125.97 deg; joints [-11.958, -63.533, 112.872, 197.274, 34.172, -116.812, -235]
  MoveL 1780 to (65.19, 25.1, -172.93) mm, rotated rx -9.61 ry -16.54 rz 125.97 deg; joints [-11.965, -63.41, 112.805, 197.24, 34.224, -116.776, -235]
  MoveL 1781 to (65.15, 23.15, -173.13) mm, rotated rx -9.61 ry -16.54 rz 125.97 deg; joints [-11.967, -63.279, 112.737, 197.207, 34.283, -116.739, -235]
  MoveL 1782 to (65.07, 21.02, -173.35) mm, rotated rx -9.61 ry -16.54 rz 125.97 deg; joints [-11.971, -63.136, 112.665, 197.171, 34.35, -116.698, -235]
  MoveL 1783 to (64.96, 18.89, -173.47) mm, rotated rx -9.61 ry -16.54 rz 125.97 deg; joints [-11.97, -62.995, 112.596, 197.141, 34.42, -116.661, -235]
  MoveL 1784 to (64.84, 16.75, -173.58) mm, rotated rx -9.61 ry -16.54 rz 125.97 deg; joints [-11.969, -62.853, 112.526, 197.112, 34.49, -116.625, -235]
  MoveL 1785 to (64.75, 14.62, -173.81) mm, rotated rx -9.61 ry -16.54 rz 125.97 deg; joints [-11.973, -62.71, 112.454, 197.075, 34.557, -116.584, -235]
  MoveL 1786 to (64.63, 12.49, -173.93) mm, rotated rx -9.61 ry -16.54 rz 125.97 deg; joints [-11.972, -62.568, 112.385, 197.046, 34.626, -116.547, -235]
  MoveL 1787 to (64.51, 10.36, -174.05) mm, rotated rx -9.61 ry -16.54 rz 125.97 deg; joints [-11.971, -62.427, 112.315, 197.016, 34.695, -116.511, -235]
  MoveL 1788 to (64.39, 8.22, -174.29) mm, rotated rx -9.61 ry -16.54 rz 125.97 deg; joints [-11.975, -62.284, 112.244, 196.98, 34.762, -116.47, -235]
  MoveL 1789 to (64.26, 6.09, -174.41) mm, rotated rx -9.61 ry -16.54 rz 125.97 deg; joints [-11.975, -62.143, 112.174, 196.951, 34.83, -116.434, -235]
  MoveL 1790 to (64.13, 3.96, -174.53) mm, rotated rx -9.61 ry -16.54 rz 125.97 deg; joints [-11.974, -62.001, 112.104, 196.922, 34.899, -116.398, -235]
  MoveL 1791 to (64.01, 1.95, -174.72) mm, rotated rx -9.61 ry -16.54 rz 125.97 deg; joints [-11.977, -61.867, 112.037, 196.89, 34.963, -116.362, -235]
  MoveL 1792 to (63.89, 0.13, -174.94) mm, rotated rx -9.61 ry -16.54 rz 125.97 deg; joints [-11.981, -61.745, 111.976, 196.858, 35.02, -116.326, -235]
  MoveL 1793 to (63.76, -1.83, -175.04) mm, rotated rx -9.61 ry -16.54 rz 125.97 deg; joints [-11.98, -61.616, 111.911, 196.832, 35.082, -116.294, -235]
  MoveL 1794 to (63.73, -4, -175.04) mm, rotated rx -9.61 ry -16.54 rz 125.97 deg; joints [-11.974, -61.471, 111.832, 196.815, 35.147, -116.268, -235]
  MoveL 1795 to (63.53, -6.72, -175.13) mm, rotated rx -9.61 ry -16.54 rz 125.97 deg; joints [-11.971, -61.291, 111.744, 196.783, 35.234, -116.225, -235]
  MoveL 1796 to (63.25, -9.16, -175.37) mm, rotated rx -9.61 ry -16.54 rz 125.97 deg; joints [-11.975, -61.13, 111.67, 196.74, 35.318, -116.177, -235]
  MoveL 1797 to (63.1, -11.19, -175.55) mm, rotated rx -9.61 ry -16.54 rz 125.97 deg; joints [-11.977, -60.995, 111.602, 196.71, 35.382, -116.142, -235]
  MoveL 1798 to (62.95, -13.06, -175.87) mm, rotated rx -9.61 ry -16.54 rz 125.97 deg; joints [-11.986, -60.87, 111.539, 196.671, 35.439, -116.102, -235]
  MoveL 1799 to (62.79, -15.1, -176.05) mm, rotated rx -9.61 ry -16.54 rz 125.97 deg; joints [-11.988, -60.735, 111.471, 196.64, 35.503, -116.067, -235]
  MoveL 1800 to (62.62, -17.06, -176.25) mm, rotated rx -9.61 ry -16.54 rz 125.97 deg; joints [-11.991, -60.604, 111.406, 196.609, 35.565, -116.031, -235]
  MoveL 1801 to (62.42, -18.98, -176.54) mm, rotated rx -9.61 ry -16.54 rz 125.97 deg; joints [-11.998, -60.477, 111.344, 196.571, 35.627, -115.992, -235]
  MoveL 1802 to (61.83, -19.67, -177.3) mm, rotated rx -9.61 ry -16.54 rz 125.97 deg; joints [-12.03, -60.434, 111.355, 196.499, 35.672, -115.933, -235]
  MoveL 1803 to (61.66, -19.34, -177.68) mm, rotated rx -9.61 ry -16.54 rz 125.97 deg; joints [-12.047, -60.456, 111.376, 196.471, 35.668, -115.915, -235]
  MoveL 1804 to (61.6, -19.28, -177.93) mm, rotated rx -9.61 ry -16.54 rz 125.97 deg; joints [-12.057, -60.46, 111.38, 196.454, 35.667, -115.904, -235]
  MoveL 1805 to (61.66, -19.48, -178.05) mm, rotated rx -9.61 ry -16.54 rz 125.97 deg; joints [-12.062, -60.444, 111.367, 196.447, 35.668, -115.899, -235]
  MoveL 1806 to (61.87, -19.96, -178.1) mm, rotated rx -9.61 ry -16.54 rz 125.97 deg; joints [-12.061, -60.409, 111.331, 196.447, 35.668, -115.899, -235]
  MoveL 1807 to (62.17, -20.56, -178.14) mm, rotated rx -9.61 ry -16.54 rz 125.97 deg; joints [-12.06, -60.364, 111.284, 196.451, 35.666, -115.902, -235]
  MoveL 1808 to (62.96, -21.92, -178.14) mm, rotated rx -9.61 ry -16.54 rz 125.97 deg; joints [-12.052, -60.262, 111.169, 196.468, 35.655, -115.916, -235]
  MoveL 1809 to (63.23, -22.39, -178.15) mm, rotated rx -9.61 ry -16.54 rz 125.97 deg; joints [-12.05, -60.227, 111.129, 196.473, 35.651, -115.921, -235]
  MoveL 1810 to (63.48, -22.86, -178.17) mm, rotated rx -9.61 ry -16.54 rz 125.97 deg; joints [-12.048, -60.192, 111.091, 196.477, 35.648, -115.924, -235]
  MoveL 1811 to (63.73, -23.35, -178.22) mm, rotated rx -9.61 ry -16.54 rz 125.97 deg; joints [-12.048, -60.155, 111.051, 196.479, 35.646, -115.926, -235]
  MoveL 1812 to (63.97, -23.86, -178.29) mm, rotated rx -9.61 ry -16.54 rz 125.97 deg; joints [-12.048, -60.117, 111.012, 196.479, 35.644, -115.926, -235]
  MoveL 1813 to (64.21, -24.36, -178.35) mm, rotated rx -9.61 ry -16.54 rz 125.97 deg; joints [-12.048, -60.08, 110.973, 196.48, 35.642, -115.927, -235]
  MoveL 1814 to (64.45, -24.79, -178.37) mm, rotated rx -9.61 ry -16.54 rz 125.97 deg; joints [-12.047, -60.047, 110.937, 196.484, 35.639, -115.93, -235]
  MoveL 1815 to (64.67, -25.19, -178.39) mm, rotated rx -9.61 ry -16.54 rz 125.97 deg; joints [-12.045, -60.018, 110.904, 196.487, 35.637, -115.933, -235]
  MoveL 1816 to (65.46, -26.55, -178.39) mm, rotated rx -9.61 ry -16.54 rz 125.97 deg; joints [-12.038, -59.916, 110.789, 196.505, 35.625, -115.948, -235]
  MoveL 1817 to (65.71, -27.01, -178.4) mm, rotated rx -9.61 ry -16.54 rz 125.97 deg; joints [-12.036, -59.882, 110.751, 196.509, 35.622, -115.952, -235]
  MoveL 1818 to (65.93, -27.43, -178.43) mm, rotated rx -9.61 ry -16.54 rz 125.97 deg; joints [-12.035, -59.85, 110.716, 196.512, 35.619, -115.954, -235]
  MoveL 1819 to (66.13, -27.83, -178.48) mm, rotated rx -9.61 ry -16.54 rz 125.97 deg; joints [-12.035, -59.82, 110.685, 196.513, 35.618, -115.955, -235]
  MoveL 1820 to (66.33, -28.23, -178.52) mm, rotated rx -9.61 ry -16.54 rz 125.97 deg; joints [-12.034, -59.79, 110.652, 196.515, 35.616, -115.957, -235]
  MoveL 1821 to (66.57, -28.66, -178.53) mm, rotated rx -9.61 ry -16.54 rz 125.97 deg; joints [-12.032, -59.758, 110.617, 196.519, 35.612, -115.96, -235]
  MoveL 1822 to (66.83, -29.11, -178.53) mm, rotated rx -9.61 ry -16.54 rz 125.97 deg; joints [-12.03, -59.724, 110.578, 196.525, 35.608, -115.965, -235]
  MoveL 1823 to (68.05, -31.78, -178.87) mm, rotated rx -9.61 ry -16.54 rz 125.97 deg; joints [-12.031, -59.527, 110.373, 196.527, 35.601, -115.968, -235]
  MoveL 1824 to (68.37, -33.06, -179.29) mm, rotated rx -9.61 ry -16.54 rz 125.97 deg; joints [-12.042, -59.434, 110.292, 196.503, 35.61, -115.95, -235]
  MoveL 1825 to (68.49, -34.3, -179.88) mm, rotated rx -9.61 ry -16.54 rz 125.97 deg; joints [-12.062, -59.346, 110.226, 196.462, 35.627, -115.919, -235]
  MoveL 1826 to (68.17, -36.66, -181.57) mm, rotated rx -9.61 ry -16.54 rz 125.97 deg; joints [-12.125, -59.182, 110.137, 196.332, 35.688, -115.818, -235]
  MoveL 1827 to (67.08, -38.87, -183.93) mm, rotated rx -9.61 ry -16.54 rz 125.97 deg; joints [-12.218, -59.035, 110.106, 196.136, 35.783, -115.666, -235]
  MoveL 1828 to (65.63, -40.37, -186.3) mm, rotated rx -9.61 ry -16.54 rz 125.97 deg; joints [-12.315, -58.939, 110.13, 195.933, 35.882, -115.509, -235]
  MoveL 1829 to (64.93, -40.65, -187.23) mm, rotated rx -9.61 ry -16.54 rz 125.97 deg; joints [-12.355, -58.924, 110.162, 195.852, 35.92, -115.446, -235]
  MoveL 1830 to (64.25, -40.61, -187.98) mm, rotated rx -9.61 ry -16.54 rz 125.97 deg; joints [-12.388, -58.931, 110.208, 195.783, 35.952, -115.394, -235]
  MoveL 1831 to (63.91, -40.47, -188.3) mm, rotated rx -9.61 ry -16.54 rz 125.97 deg; joints [-12.403, -58.943, 110.236, 195.753, 35.965, -115.371, -235]
  MoveL 1832 to (63.57, -40.25, -188.58) mm, rotated rx -9.61 ry -16.54 rz 125.97 deg; joints [-12.416, -58.96, 110.268, 195.726, 35.977, -115.351, -235]
  MoveL 1833 to (62.92, -39.58, -189) mm, rotated rx -9.61 ry -16.54 rz 125.97 deg; joints [-12.438, -59.011, 110.341, 195.682, 35.995, -115.318, -235]
  MoveL 1834 to (62.28, -38.59, -189.25) mm, rotated rx -9.61 ry -16.54 rz 125.97 deg; joints [-12.454, -59.084, 110.428, 195.651, 36.005, -115.295, -235]
  MoveL 1835 to (61.65, -37.29, -189.34) mm, rotated rx -9.61 ry -16.54 rz 125.97 deg; joints [-12.465, -59.179, 110.528, 195.633, 36.008, -115.282, -235]
  MoveL 1836 to (61.04, -35.84, -189.34) mm, rotated rx -9.61 ry -16.54 rz 125.97 deg; joints [-12.472, -59.284, 110.634, 195.621, 36.008, -115.274, -235]
  MoveL 1837 to (60.84, -35.35, -189.33) mm, rotated rx -9.61 ry -16.54 rz 125.97 deg; joints [-12.474, -59.32, 110.67, 195.617, 36.008, -115.272, -235]
  MoveL 1838 to (60.64, -34.81, -189.3) mm, rotated rx -9.61 ry -16.54 rz 125.97 deg; joints [-12.476, -59.359, 110.707, 195.616, 36.006, -115.271, -235]
  MoveL 1839 to (60.43, -34.2, -189.23) mm, rotated rx -9.61 ry -16.54 rz 125.97 deg; joints [-12.476, -59.403, 110.749, 195.616, 36.003, -115.273, -235]
  MoveL 1840 to (60.23, -33.67, -189.21) mm, rotated rx -9.61 ry -16.54 rz 125.97 deg; joints [-12.477, -59.441, 110.786, 195.614, 36.002, -115.271, -235]
  MoveL 1841 to (60.03, -33.19, -189.2) mm, rotated rx -9.61 ry -16.54 rz 125.97 deg; joints [-12.48, -59.477, 110.821, 195.61, 36.002, -115.269, -235]
  MoveL 1842 to (59.83, -32.71, -189.19) mm, rotated rx -9.61 ry -16.54 rz 125.97 deg; joints [-12.482, -59.511, 110.856, 195.607, 36.001, -115.267, -235]
  MoveL 1843 to (59.66, -32.22, -189.15) mm, rotated rx -9.61 ry -16.54 rz 125.97 deg; joints [-12.482, -59.546, 110.889, 195.607, 35.999, -115.268, -235]
  MoveL 1844 to (59.52, -31.75, -189.07) mm, rotated rx -9.61 ry -16.54 rz 125.97 deg; joints [-12.481, -59.581, 110.92, 195.61, 35.996, -115.27, -235]
  MoveL 1845 to (59.38, -31.26, -188.97) mm, rotated rx -9.61 ry -16.54 rz 125.97 deg; joints [-12.479, -59.616, 110.951, 195.615, 35.993, -115.274, -235]
  MoveL 1846 to (59.23, -30.77, -188.9) mm, rotated rx -9.61 ry -16.54 rz 125.97 deg; joints [-12.479, -59.651, 110.984, 195.617, 35.99, -115.276, -235]
  MoveL 1847 to (59.04, -30.27, -188.87) mm, rotated rx -9.61 ry -16.54 rz 125.97 deg; joints [-12.48, -59.687, 111.018, 195.615, 35.989, -115.275, -235]
  MoveL 1848 to (58.85, -29.79, -188.86) mm, rotated rx -9.61 ry -16.54 rz 125.97 deg; joints [-12.482, -59.722, 111.053, 195.612, 35.988, -115.273, -235]
  MoveL 1849 to (57.89, -27.42, -188.85) mm, rotated rx -9.61 ry -16.54 rz 125.97 deg; joints [-12.493, -59.894, 111.221, 195.595, 35.983, -115.263, -235]
  MoveL 1850 to (57.8, -27.04, -188.83) mm, rotated rx -9.61 ry -16.54 rz 125.97 deg; joints [-12.494, -59.921, 111.244, 195.595, 35.978, -115.264, -235]
  MoveL 1851 to (57.78, -26.88, -188.71) mm, rotated rx -9.61 ry -16.54 rz 125.97 deg; joints [-12.49, -59.933, 111.253, 195.603, 35.976, -115.27, -235]
  MoveL 1852 to (57.8, -26.96, -188.48) mm, rotated rx -9.61 ry -16.54 rz 125.97 deg; joints [-12.48, -59.928, 111.251, 195.618, 35.98, -115.279, -235]
  MoveL 1853 to (57.86, -27.32, -188.12) mm, rotated rx -9.61 ry -16.54 rz 125.97 deg; joints [-12.464, -59.906, 111.237, 195.641, 35.991, -115.291, -235]
  MoveL 1854 to (58.39, -26.76, -187.38) mm, rotated rx -9.61 ry -16.54 rz 125.97 deg; joints [-12.433, -59.941, 111.226, 195.707, 35.952, -115.344, -235]
  MoveL 1855 to (58.8, -24.68, -187.36) mm, rotated rx -9.61 ry -16.54 rz 125.97 deg; joints [-12.437, -60.075, 111.277, 195.732, 35.871, -115.379, -235]
  MoveL 1856 to (59.24, -22.54, -187.23) mm, rotated rx -9.61 ry -16.54 rz 125.97 deg; joints [-12.436, -60.213, 111.327, 195.767, 35.787, -115.42, -235]
  MoveL 1857 to (59.74, -20.33, -186.97) mm, rotated rx -9.61 ry -16.54 rz 125.97 deg; joints [-12.43, -60.357, 111.378, 195.812, 35.699, -115.469, -235]
  MoveL 1858 to (60.18, -18.25, -186.84) mm, rotated rx -9.61 ry -16.54 rz 125.97 deg; joints [-12.429, -60.49, 111.426, 195.846, 35.617, -115.511, -235]
  MoveL 1859 to (60.61, -16.25, -186.58) mm, rotated rx -9.61 ry -16.54 rz 125.97 deg; joints [-12.422, -60.62, 111.474, 195.888, 35.539, -115.556, -235]
  MoveL 1860 to (61.06, -14.2, -186.22) mm, rotated rx -9.61 ry -16.54 rz 125.97 deg; joints [-12.412, -60.754, 111.522, 195.938, 35.458, -115.607, -235]
  MoveL 1861 to (61.49, -12.09, -186.09) mm, rotated rx -9.61 ry -16.54 rz 125.97 deg; joints [-12.411, -60.889, 111.571, 195.973, 35.375, -115.65, -235]
  MoveL 1862 to (61.9, -10.02, -185.99) mm, rotated rx -9.61 ry -16.54 rz 125.97 deg; joints [-12.411, -61.023, 111.619, 196.006, 35.293, -115.69, -235]
  MoveL 1863 to (62.32, -7.91, -185.84) mm, rotated rx -9.61 ry -16.54 rz 125.97 deg; joints [-12.409, -61.159, 111.669, 196.042, 35.21, -115.733, -235]
  MoveL 1864 to (62.75, -5.87, -185.55) mm, rotated rx -9.61 ry -16.54 rz 125.97 deg; joints [-12.402, -61.291, 111.716, 196.088, 35.13, -115.782, -235]
  MoveL 1865 to (63.13, -3.72, -185.21) mm, rotated rx -9.61 ry -16.54 rz 125.97 deg; joints [-12.393, -61.432, 111.771, 196.137, 35.049, -115.833, -235]
  MoveL 1866 to (63.53, -1.63, -185.03) mm, rotated rx -9.61 ry -16.54 rz 125.97 deg; joints [-12.39, -61.567, 111.821, 196.175, 34.968, -115.878, -235]
  MoveL 1867 to (63.92, 0.48, -184.92) mm, rotated rx -9.61 ry -16.54 rz 125.97 deg; joints [-12.39, -61.703, 111.87, 196.21, 34.885, -115.92, -235]
  MoveL 1868 to (64.32, 2.56, -184.85) mm, rotated rx -9.61 ry -16.54 rz 125.97 deg; joints [-12.392, -61.837, 111.918, 196.242, 34.801, -115.96, -235]
  MoveL 1869 to (64.7, 4.67, -184.63) mm, rotated rx -9.61 ry -16.54 rz 125.97 deg; joints [-12.387, -61.974, 111.969, 196.284, 34.72, -116.007, -235]
  MoveL 1870 to (65.08, 6.76, -184.49) mm, rotated rx -9.61 ry -16.54 rz 125.97 deg; joints [-12.386, -62.109, 112.017, 196.321, 34.637, -116.051, -235]
  MoveL 1871 to (65.48, 8.87, -184.41) mm, rotated rx -9.61 ry -16.54 rz 125.97 deg; joints [-12.387, -62.244, 112.065, 196.354, 34.552, -116.093, -235]
  MoveL 1872 to (65.84, 10.96, -184.18) mm, rotated rx -9.61 ry -16.54 rz 125.97 deg; joints [-12.383, -62.38, 112.116, 196.397, 34.472, -116.14, -235]
  MoveL 1873 to (66.19, 13.08, -183.95) mm, rotated rx -9.61 ry -16.54 rz 125.97 deg; joints [-12.378, -62.518, 112.168, 196.44, 34.39, -116.189, -235]
  MoveL 1874 to (66.57, 15.23, -183.8) mm, rotated rx -9.61 ry -16.54 rz 125.97 deg; joints [-12.377, -62.657, 112.218, 196.48, 34.306, -116.235, -235]
  MoveL 1875 to (66.86, 17.09, -183.68) mm, rotated rx -9.61 ry -16.54 rz 125.97 deg; joints [-12.376, -62.777, 112.263, 196.512, 34.234, -116.273, -235]
  MoveL 1876 to (67.06, 18.71, -183.47) mm, rotated rx -9.61 ry -16.54 rz 125.97 deg; joints [-12.371, -62.884, 112.309, 196.545, 34.176, -116.31, -235]
  MoveL 1877 to (67.16, 20.15, -183.14) mm, rotated rx -9.61 ry -16.54 rz 125.97 deg; joints [-12.362, -62.98, 112.356, 196.582, 34.131, -116.345, -235]
  MoveL 1878 to (66.66, 18.76, -182.19) mm, rotated rx -9.61 ry -16.54 rz 125.97 deg; joints [-12.321, -62.902, 112.357, 196.618, 34.214, -116.35, -235]
  MoveL 1879 to (66.75, 19.25, -182.19) mm, rotated rx -9.61 ry -16.54 rz 125.97 deg; joints [-12.322, -62.933, 112.367, 196.625, 34.194, -116.36, -235]
  MoveL 1880 to (66.89, 19.73, -182.18) mm, rotated rx -9.61 ry -16.54 rz 125.97 deg; joints [-12.322, -62.963, 112.373, 196.634, 34.171, -116.371, -235]
  MoveL 1881 to (67.12, 20.21, -182.16) mm, rotated rx -9.61 ry -16.54 rz 125.97 deg; joints [-12.322, -62.991, 112.372, 196.647, 34.143, -116.387, -235]
  MoveL 1882 to (67.42, 20.68, -182.12) mm, rotated rx -9.61 ry -16.54 rz 125.97 deg; joints [-12.32, -63.019, 112.366, 196.664, 34.111, -116.406, -235]
  MoveL 1883 to (67.79, 21.17, -182.06) mm, rotated rx -9.61 ry -16.54 rz 125.97 deg; joints [-12.317, -63.046, 112.355, 196.685, 34.075, -116.428, -235]
  MoveL 1884 to (68.18, 21.6, -182.02) mm, rotated rx -9.61 ry -16.54 rz 125.97 deg; joints [-12.315, -63.069, 112.34, 196.704, 34.04, -116.45, -235]
  MoveL 1885 to (68.57, 22.01, -182.01) mm, rotated rx -9.61 ry -16.54 rz 125.97 deg; joints [-12.314, -63.09, 112.324, 196.722, 34.004, -116.47, -235]
  MoveL 1886 to (68.94, 22.38, -182.01) mm, rotated rx -9.61 ry -16.54 rz 125.97 deg; joints [-12.313, -63.109, 112.309, 196.738, 33.971, -116.489, -235]
  MoveL 1887 to (69.3, 22.76, -182) mm, rotated rx -9.61 ry -16.54 rz 125.97 deg; joints [-12.313, -63.128, 112.293, 196.754, 33.938, -116.508, -235]
  MoveL 1888 to (69.7, 23.2, -181.96) mm, rotated rx -9.61 ry -16.54 rz 125.97 deg; joints [-12.31, -63.151, 112.278, 196.774, 33.902, -116.53, -235]
  MoveL 1889 to (70.11, 23.71, -181.87) mm, rotated rx -9.61 ry -16.54 rz 125.97 deg; joints [-12.306, -63.179, 112.264, 196.799, 33.863, -116.556, -235]
  MoveL 1890 to (70.45, 24.1, -181.82) mm, rotated rx -9.61 ry -16.54 rz 125.97 deg; joints [-12.304, -63.2, 112.252, 196.817, 33.831, -116.576, -235]
  MoveL 1891 to (70.74, 24.41, -181.8) mm, rotated rx -9.61 ry -16.54 rz 125.97 deg; joints [-12.302, -63.216, 112.24, 196.832, 33.805, -116.592, -235]
  MoveL 1892 to (71.08, 24.76, -181.78) mm, rotated rx -9.61 ry -16.54 rz 125.97 deg; joints [-12.301, -63.234, 112.226, 196.848, 33.775, -116.61, -235]
  MoveL 1893 to (71.44, 25.13, -181.78) mm, rotated rx -9.61 ry -16.54 rz 125.97 deg; joints [-12.301, -63.253, 112.21, 196.864, 33.742, -116.629, -235]
  MoveL 1894 to (71.79, 25.49, -181.77) mm, rotated rx -9.61 ry -16.54 rz 125.97 deg; joints [-12.3, -63.272, 112.196, 196.88, 33.71, -116.648, -235]
  MoveL 1895 to (72.13, 25.86, -181.74) mm, rotated rx -9.61 ry -16.54 rz 125.97 deg; joints [-12.298, -63.291, 112.182, 196.897, 33.679, -116.667, -235]
  MoveL 1896 to (72.49, 26.23, -181.73) mm, rotated rx -9.61 ry -16.54 rz 125.97 deg; joints [-12.297, -63.309, 112.167, 196.914, 33.647, -116.686, -235]
  MoveL 1897 to (74.34, 28.1, -181.73) mm, rotated rx -9.61 ry -16.54 rz 125.97 deg; joints [-12.294, -63.403, 112.086, 196.996, 33.48, -116.781, -235]
  MoveL 1898 to (75.4, 29.08, -181.81) mm, rotated rx -9.61 ry -16.54 rz 125.97 deg; joints [-12.295, -63.45, 112.035, 197.037, 33.386, -116.832, -235]
  MoveL 1899 to (76.38, 29.79, -182.06) mm, rotated rx -9.61 ry -16.54 rz 125.97 deg; joints [-12.303, -63.479, 111.979, 197.061, 33.304, -116.868, -235]
  MoveL 1900 to (77.25, 30.2, -182.48) mm, rotated rx -9.61 ry -16.54 rz 125.97 deg; joints [-12.317, -63.489, 111.919, 197.068, 33.234, -116.889, -235]
  MoveL 1901 to (78.02, 30.34, -183.06) mm, rotated rx -9.61 ry -16.54 rz 125.97 deg; joints [-12.338, -63.481, 111.856, 197.058, 33.177, -116.895, -235]
  MoveL 1902 to (78.7, 30.19, -183.81) mm, rotated rx -9.61 ry -16.54 rz 125.97 deg; joints [-12.365, -63.455, 111.788, 197.03, 33.132, -116.886, -235]
  MoveL 1903 to (79.28, 29.76, -184.72) mm, rotated rx -9.61 ry -16.54 rz 125.97 deg; joints [-12.398, -63.41, 111.715, 196.984, 33.099, -116.861, -235]
  MoveL 1904 to (80.15, 28.05, -187.06) mm, rotated rx -9.61 ry -16.54 rz 125.97 deg; joints [-12.484, -63.265, 111.559, 196.842, 33.071, -116.767, -235]
  MoveL 1905 to (80.44, 25.79, -189.4) mm, rotated rx -9.61 ry -16.54 rz 125.97 deg; joints [-12.572, -63.094, 111.428, 196.673, 33.093, -116.644, -235]
  MoveL 1906 to (79.97, 23.57, -191.11) mm, rotated rx -9.61 ry -16.54 rz 125.97 deg; joints [-12.637, -62.943, 111.366, 196.522, 33.166, -116.522, -235]
  MoveL 1907 to (79.46, 22.48, -191.72) mm, rotated rx -9.61 ry -16.54 rz 125.97 deg; joints [-12.661, -62.874, 111.36, 196.453, 33.222, -116.461, -235]
  MoveL 1908 to (78.75, 21.39, -192.18) mm, rotated rx -9.61 ry -16.54 rz 125.97 deg; joints [-12.68, -62.811, 111.372, 196.389, 33.29, -116.401, -235]
  MoveL 1909 to (76.78, 19.25, -192.61) mm, rotated rx -9.61 ry -16.54 rz 125.97 deg; joints [-12.7, -62.698, 111.447, 196.273, 33.467, -116.281, -235]
  MoveL 1910 to (76.03, 18.57, -192.64) mm, rotated rx -9.61 ry -16.54 rz 125.97 deg; joints [-12.703, -62.666, 111.482, 196.24, 33.531, -116.243, -235]
  MoveL 1911 to (73.96, 16.96, -192.64) mm, rotated rx -9.61 ry -16.54 rz 125.97 deg; joints [-12.708, -62.592, 111.588, 196.156, 33.703, -116.147, -235]
  MoveL 1912 to (73.2, 16.31, -192.7) mm, rotated rx -9.61 ry -16.54 rz 125.97 deg; joints [-12.712, -62.561, 111.625, 196.121, 33.767, -116.109, -235]
  MoveL 1913 to (72.37, 15.66, -192.7) mm, rotated rx -9.61 ry -16.54 rz 125.97 deg; joints [-12.714, -62.531, 111.667, 196.087, 33.836, -116.07, -235]
  MoveL 1914 to (71.99, 15.36, -192.71) mm, rotated rx -9.61 ry -16.54 rz 125.97 deg; joints [-12.716, -62.517, 111.686, 196.071, 33.867, -116.053, -235]
  MoveL 1915 to (71.66, 15.08, -192.73) mm, rotated rx -9.61 ry -16.54 rz 125.97 deg; joints [-12.717, -62.504, 111.702, 196.057, 33.895, -116.036, -235]
  MoveL 1916 to (71.3, 14.79, -192.74) mm, rotated rx -9.61 ry -16.54 rz 125.97 deg; joints [-12.719, -62.49, 111.719, 196.041, 33.925, -116.019, -235]
  MoveL 1917 to (69.24, 13.18, -192.75) mm, rotated rx -9.61 ry -16.54 rz 125.97 deg; joints [-12.724, -62.415, 111.824, 195.959, 34.096, -115.925, -235]
  MoveL 1918 to (68.86, 12.86, -192.77) mm, rotated rx -9.61 ry -16.54 rz 125.97 deg; joints [-12.725, -62.4, 111.842, 195.943, 34.128, -115.907, -235]
  MoveL 1919 to (68.52, 12.54, -192.81) mm, rotated rx -9.61 ry -16.54 rz 125.97 deg; joints [-12.728, -62.384, 111.857, 195.927, 34.157, -115.889, -235]
  MoveL 1920 to (68.22, 12.22, -192.85) mm, rotated rx -9.61 ry -16.54 rz 125.97 deg; joints [-12.73, -62.367, 111.868, 195.912, 34.184, -115.873, -235]
  MoveL 1921 to (67.95, 11.88, -192.88) mm, rotated rx -9.61 ry -16.54 rz 125.97 deg; joints [-12.731, -62.348, 111.877, 195.898, 34.21, -115.858, -235]
  MoveL 1922 to (67.73, 11.5, -192.9) mm, rotated rx -9.61 ry -16.54 rz 125.97 deg; joints [-12.732, -62.326, 111.88, 195.887, 34.234, -115.845, -235]
  MoveL 1923 to (67.55, 11.09, -192.9) mm, rotated rx -9.61 ry -16.54 rz 125.97 deg; joints [-12.732, -62.302, 111.879, 195.878, 34.257, -115.834, -235]
  MoveL 1924 to (67.98, 11.72, -193.64) mm, rotated rx -9.61 ry -16.54 rz 125.97 deg; joints [-12.762, -62.332, 111.859, 195.847, 34.204, -115.825, -235]
  MoveL 1925 to (67.78, 10.3, -194.19) mm, rotated rx -9.61 ry -16.54 rz 125.97 deg; joints [-12.781, -62.236, 111.817, 195.794, 34.251, -115.778, -235]
  MoveL 1926 to (67.46, 8.78, -194.62) mm, rotated rx -9.61 ry -16.54 rz 125.97 deg; joints [-12.795, -62.136, 111.78, 195.746, 34.31, -115.732, -235]
  MoveL 1927 to (67.02, 7.06, -194.92) mm, rotated rx -9.61 ry -16.54 rz 125.97 deg; joints [-12.804, -62.027, 111.748, 195.699, 34.383, -115.684, -235]
  MoveL 1928 to (66.43, 5.13, -195.11) mm, rotated rx -9.61 ry -16.54 rz 125.97 deg; joints [-12.808, -61.905, 111.721, 195.655, 34.473, -115.635, -235]
  MoveL 1929 to (65.82, 3.12, -195.3) mm, rotated rx -9.61 ry -16.54 rz 125.97 deg; joints [-12.813, -61.779, 111.693, 195.609, 34.566, -115.583, -235]
  MoveL 1930 to (65.17, 1.09, -195.42) mm, rotated rx -9.61 ry -16.54 rz 125.97 deg; joints [-12.814, -61.653, 111.667, 195.568, 34.663, -115.534, -235]
  MoveL 1931 to (64.53, -0.94, -195.65) mm, rotated rx -9.61 ry -16.54 rz 125.97 deg; joints [-12.82, -61.525, 111.638, 195.52, 34.758, -115.481, -235]
  MoveL 1932 to (63.87, -2.97, -195.76) mm, rotated rx -9.61 ry -16.54 rz 125.97 deg; joints [-12.822, -61.398, 111.612, 195.479, 34.854, -115.432, -235]
  MoveL 1933 to (63.21, -5, -195.88) mm, rotated rx -9.61 ry -16.54 rz 125.97 deg; joints [-12.823, -61.271, 111.586, 195.438, 34.951, -115.384, -235]
  MoveL 1934 to (62.55, -7.03, -196) mm, rotated rx -9.61 ry -16.54 rz 125.97 deg; joints [-12.825, -61.144, 111.559, 195.397, 35.047, -115.336, -235]
  MoveL 1935 to (61.89, -9.06, -196.23) mm, rotated rx -9.61 ry -16.54 rz 125.97 deg; joints [-12.831, -61.017, 111.531, 195.35, 35.142, -115.283, -235]
  MoveL 1936 to (61.23, -11.09, -196.35) mm, rotated rx -9.61 ry -16.54 rz 125.97 deg; joints [-12.832, -60.89, 111.504, 195.309, 35.238, -115.236, -235]
  MoveL 1937 to (60.64, -13.06, -196.46) mm, rotated rx -9.61 ry -16.54 rz 125.97 deg; joints [-12.833, -60.766, 111.472, 195.274, 35.327, -115.193, -235]
  MoveL 1938 to (60.18, -15.02, -196.66) mm, rotated rx -9.61 ry -16.54 rz 125.97 deg; joints [-12.838, -60.64, 111.431, 195.235, 35.408, -115.15, -235]
  MoveL 1939 to (59.37, -17.38, -196.8) mm, rotated rx -9.61 ry -16.54 rz 125.97 deg; joints [-12.84, -60.491, 111.4, 195.189, 35.521, -115.094, -235]
  MoveL 1940 to (58.46, -19.66, -196.88) mm, rotated rx -9.61 ry -16.54 rz 125.97 deg; joints [-12.84, -60.351, 111.382, 195.143, 35.639, -115.039, -235]
  MoveL 1941 to (57.67, -21.81, -196.92) mm, rotated rx -9.61 ry -16.54 rz 125.97 deg; joints [-12.838, -60.218, 111.359, 195.106, 35.746, -114.991, -235]
  MoveL 1942 to (57.01, -23.75, -196.96) mm, rotated rx -9.61 ry -16.54 rz 125.97 deg; joints [-12.837, -60.096, 111.333, 195.073, 35.839, -114.95, -235]
  MoveL 1943 to (56.39, -25.61, -197.08) mm, rotated rx -9.61 ry -16.54 rz 125.97 deg; joints [-12.839, -59.979, 111.307, 195.037, 35.926, -114.908, -235]
  MoveL 1944 to (55.76, -27.53, -197.14) mm, rotated rx -9.61 ry -16.54 rz 125.97 deg; joints [-12.839, -59.858, 111.28, 195.005, 36.016, -114.867, -235]
  MoveL 1945 to (55.08, -29.55, -197.22) mm, rotated rx -9.61 ry -16.54 rz 125.97 deg; joints [-12.839, -59.732, 111.251, 194.97, 36.111, -114.824, -235]
  MoveL 1946 to (54.43, -31.43, -197.4) mm, rotated rx -9.61 ry -16.54 rz 125.97 deg; joints [-12.843, -59.613, 111.225, 194.93, 36.2, -114.779, -235]
  MoveL 1947 to (53.78, -33.22, -197.71) mm, rotated rx -9.61 ry -16.54 rz 125.97 deg; joints [-12.853, -59.499, 111.2, 194.883, 36.284, -114.73, -235]
  MoveL 1948 to (53.11, -33.78, -198.75) mm, rotated rx -9.61 ry -16.54 rz 125.97 deg; joints [-12.897, -59.463, 111.215, 194.795, 36.327, -114.664, -235]
  MoveL 1949 to (53.14, -33.52, -199.27) mm, rotated rx -9.61 ry -16.54 rz 125.97 deg; joints [-12.918, -59.476, 111.217, 194.765, 36.312, -114.647, -235]
  MoveL 1950 to (53.12, -33.5, -199.59) mm, rotated rx -9.61 ry -16.54 rz 125.97 deg; joints [-12.932, -59.476, 111.215, 194.744, 36.309, -114.634, -235]
  MoveL 1951 to (53.07, -33.71, -199.76) mm, rotated rx -9.61 ry -16.54 rz 125.97 deg; joints [-12.938, -59.461, 111.208, 194.731, 36.316, -114.624, -235]
  MoveL 1952 to (53.04, -34.14, -199.79) mm, rotated rx -9.61 ry -16.54 rz 125.97 deg; joints [-12.938, -59.433, 111.193, 194.726, 36.328, -114.618, -235]
  MoveL 1953 to (53.05, -34.65, -199.81) mm, rotated rx -9.61 ry -16.54 rz 125.97 deg; joints [-12.937, -59.398, 111.171, 194.724, 36.341, -114.614, -235]
  MoveL 1954 to (53.15, -35.24, -199.82) mm, rotated rx -9.61 ry -16.54 rz 125.97 deg; joints [-12.935, -59.357, 111.14, 194.723, 36.35, -114.612, -235]
  MoveL 1955 to (53.29, -35.86, -199.83) mm, rotated rx -9.61 ry -16.54 rz 125.97 deg; joints [-12.933, -59.314, 111.104, 194.724, 36.358, -114.611, -235]
  MoveL 1956 to (54.27, -39.39, -199.83) mm, rotated rx -9.61 ry -16.54 rz 125.97 deg; joints [-12.916, -59.064, 110.885, 194.74, 36.39, -114.614, -235]
  MoveL 1957 to (54.38, -39.82, -199.86) mm, rotated rx -9.61 ry -16.54 rz 125.97 deg; joints [-12.916, -59.034, 110.86, 194.74, 36.395, -114.613, -235]
  MoveL 1958 to (54.5, -40.29, -199.87) mm, rotated rx -9.61 ry -16.54 rz 125.97 deg; joints [-12.914, -59.001, 110.831, 194.741, 36.399, -114.613, -235]
  MoveL 1959 to (54.64, -40.79, -199.88) mm, rotated rx -9.61 ry -16.54 rz 125.97 deg; joints [-12.912, -58.965, 110.8, 194.743, 36.404, -114.613, -235]
  MoveL 1960 to (54.76, -41.27, -199.89) mm, rotated rx -9.61 ry -16.54 rz 125.97 deg; joints [-12.91, -58.932, 110.771, 194.743, 36.409, -114.613, -235]
  MoveL 1961 to (54.86, -41.72, -199.93) mm, rotated rx -9.61 ry -16.54 rz 125.97 deg; joints [-12.91, -58.9, 110.744, 194.742, 36.414, -114.611, -235]
  MoveL 1962 to (54.93, -42.14, -199.99) mm, rotated rx -9.61 ry -16.54 rz 125.97 deg; joints [-12.911, -58.87, 110.72, 194.739, 36.42, -114.608, -235]
  MoveL 1963 to (55.04, -42.6, -200.03) mm, rotated rx -9.61 ry -16.54 rz 125.97 deg; joints [-12.91, -58.838, 110.693, 194.738, 36.425, -114.606, -235]
  MoveL 1964 to (55.15, -43.08, -200.04) mm, rotated rx -9.61 ry -16.54 rz 125.97 deg; joints [-12.909, -58.804, 110.665, 194.739, 36.429, -114.605, -235]
  MoveL 1965 to (55.29, -43.56, -200.05) mm, rotated rx -9.61 ry -16.54 rz 125.97 deg; joints [-12.907, -58.77, 110.634, 194.741, 36.434, -114.606, -235]
  MoveL 1966 to (55.43, -44.07, -200.05) mm, rotated rx -9.61 ry -16.54 rz 125.97 deg; joints [-12.904, -58.734, 110.603, 194.743, 36.438, -114.606, -235]
  MoveL 1967 to (55.93, -46.94, -200.39) mm, rotated rx -9.61 ry -16.54 rz 125.97 deg; joints [-12.906, -58.533, 110.442, 194.726, 36.477, -114.587, -235]
  MoveL 1968 to (55.92, -48.24, -200.83) mm, rotated rx -9.61 ry -16.54 rz 125.97 deg; joints [-12.92, -58.443, 110.384, 194.694, 36.505, -114.56, -235]
  MoveL 1969 to (55.73, -49.45, -201.43) mm, rotated rx -9.61 ry -16.54 rz 125.97 deg; joints [-12.941, -58.36, 110.34, 194.646, 36.541, -114.522, -235]
  MoveL 1970 to (54.82, -51.6, -203.16) mm, rotated rx -9.61 ry -16.54 rz 125.97 deg; joints [-13.008, -58.216, 110.299, 194.505, 36.63, -114.411, -235]
  MoveL 1971 to (53.22, -53.38, -205.59) mm, rotated rx -9.61 ry -16.54 rz 125.97 deg; joints [-13.107, -58.099, 110.318, 194.302, 36.745, -114.257, -235]
